LIN {X 0,Y 206.722,Z 761.527,A -85,B 0,C 180,E1 -21275.32,E2 -21275.32} C_VEL
LIN {X 0,Y 206.672,Z 761.479,A -85,B 0,C 180,E1 -21280.248,E2 -21280.248} C_VEL
LIN {X 0,Y 206.66,Z 761.554,A -85,B 0,C 180,E1 -21284.426,E2 -21284.426} C_VEL
LIN {X 0,Y 206.671,Z 761.526,A -85,B 0,C 180,E1 -21289.751,E2 -21289.751} C_VEL
LIN {X 0,Y 206.77,Z 761.618,A -85,B 0,C 180,E1 -21293.35,E2 -21293.35} C_VEL
LIN {X 0,Y 208.15,Z 768.058,A -85,B 0,C 180,E1 -21297.269,E2 -21297.269} C_VEL
LIN {X 0,Y 208.652,Z 770.291,A -85,B 0,C 180,E1 -21298.098,E2 -21298.098} C_VEL
LIN {X 0,Y 209.266,Z 773.35,A -85,B 0,C 180,E1 -21298.708,E2 -21298.708} C_VEL
LIN {X 0,Y 210.111,Z 778.796,A -85,B 0,C 180,E1 -21299.305,E2 -21299.305} C_VEL
LIN {X 0,Y 211.076,Z 793.394,A -85,B 0,C 180,E1 -21300.045,E2 -21300.045} C_VEL
LIN {X 0,Y 211.633,Z 797.547,A -85,B 0,C 180,E1 -21300.292,E2 -21300.292} C_VEL
LIN {X 0,Y 214.362,Z 818.731,A -85,B 0,C 180,E1 -21301.497,E2 -21301.497} C_VEL
LIN {X 0,Y 213.279,Z 848.564,A -85,B 0,C 180,E1 -21302.527,E2 -21302.527} C_VEL
LIN {X 0,Y 212.374,Z 858.849,A -85,B 0,C 180,E1 -21303.133,E2 -21303.133} C_VEL
LIN {X 0,Y 210.969,Z 869.629,A -85,B 0,C 180,E1 -21304.099,E2 -21304.099} C_VEL
LIN {X 0,Y 209.383,Z 879.305,A -85,B 0,C 180,E1 -21305.334,E2 -21305.334} C_VEL
LIN {X 0,Y 207.795,Z 887.072,A -85,B 0,C 180,E1 -21306.584,E2 -21306.584} C_VEL
LIN {X 0,Y 205.953,Z 895.137,A -85,B 0,C 180,E1 -21308.216,E2 -21308.216} C_VEL
LIN {X 0,Y 204.314,Z 901.802,A -85,B 0,C 180,E1 -21309.88,E2 -21309.88} C_VEL
LIN {X 0,Y 202.599,Z 908.13,A -85,B 0,C 180,E1 -21311.808,E2 -21311.808} C_VEL
LIN {X 0,Y 201.115,Z 913.389,A -85,B 0,C 180,E1 -21313.766,E2 -21313.766} C_VEL
LIN {X 0,Y 199.973,Z 917.78,A -85,B 0,C 180,E1 -21315.758,E2 -21315.758} C_VEL
LIN {X 0,Y 198.631,Z 922.961,A -85,B 0,C 180,E1 -21318.779,E2 -21318.779} C_VEL
LIN {X 0,Y 197.771,Z 926.768,A -85,B 0,C 180,E1 -21321.828,E2 -21321.828} C_VEL
LIN {X 0,Y 197.428,Z 928.517,A -85,B 0,C 180,E1 -21323.869,E2 -21323.869} C_VEL
LIN {X 0,Y 197.324,Z 929.773,A -85,B 0,C 180,E1 -21325.915,E2 -21325.915} C_VEL
LIN {X 0,Y 197.284,Z 930.553,A -85,B 0,C 180,E1 -21327.958,E2 -21327.958} C_VEL
LIN {X 0,Y 197.367,Z 930.849,A -85,B 0,C 180,E1 -21330,E2 -21330} C_VEL
LIN {X 0,Y 197.279,Z 930.544,A -85,B 0,C 180,E1 -21332.042,E2 -21332.042} C_VEL
LIN {X 0,Y 197.285,Z 929.748,A -85,B 0,C 180,E1 -21334.086,E2 -21334.086} C_VEL
LIN {X 0,Y 197.428,Z 928.477,A -85,B 0,C 180,E1 -21336.131,E2 -21336.131} C_VEL
LIN {X 0,Y 197.996,Z 925.55,A -85,B 0,C 180,E1 -21339.191,E2 -21339.191} C_VEL
LIN {X 0,Y 198.63,Z 922.885,A -85,B 0,C 180,E1 -21341.222,E2 -21341.222} C_VEL
LIN {X 0,Y 199.97,Z 917.682,A -85,B 0,C 180,E1 -21344.242,E2 -21344.242} C_VEL
LIN {X 0,Y 201.813,Z 910.825,A -85,B 0,C 180,E1 -21347.218,E2 -21347.218} C_VEL
LIN {X 0,Y 203.836,Z 903.341,A -85,B 0,C 180,E1 -21349.644,E2 -21349.644} C_VEL
LIN {X 0,Y 205.695,Z 895.961,A -85,B 0,C 180,E1 -21351.549,E2 -21351.549} C_VEL
LIN {X 0,Y 207.524,Z 888.058,A -85,B 0,C 180,E1 -21353.184,E2 -21353.184} C_VEL
LIN {X 0,Y 209.302,Z 879.229,A -85,B 0,C 180,E1 -21354.637,E2 -21354.637} C_VEL
LIN {X 0,Y 211.087,Z 868.011,A -85,B 0,C 180,E1 -21356.031,E2 -21356.031} C_VEL
LIN {X 0,Y 212.469,Z 857.353,A -85,B 0,C 180,E1 -21356.92,E2 -21356.92} C_VEL
LIN {X 0,Y 213.257,Z 847.507,A -85,B 0,C 180,E1 -21357.476,E2 -21357.476} C_VEL
LIN {X 0,Y 214.211,Z 817.801,A -85,B 0,C 180,E1 -21358.505,E2 -21358.505} C_VEL
LIN {X 0,Y 211.265,Z 795.967,A -85,B 0,C 180,E1 -21359.768,E2 -21359.768} C_VEL
LIN {X 0,Y 210.289,Z 791.346,A -85,B 0,C 180,E1 -21360.097,E2 -21360.097} C_VEL
LIN {X 0,Y 204.304,Z 777.141,A -85,B 0,C 180,E1 -21361.637,E2 -21361.637} C_VEL
LIN {X 0,Y 201.519,Z 770.64,A -85,B 0,C 180,E1 -21362.466,E2 -21362.466} C_VEL
LIN {X 0,Y 200.877,Z 767.771,A -85,B 0,C 180,E1 -21364.041,E2 -21364.041} C_VEL
LIN {X 0,Y 199.699,Z 762.434,A -85,B 0,C 180,E1 -21367.537,E2 -21367.537} C_VEL
LIN {X 0,Y 199.577,Z 762.407,A -85,B 0,C 180,E1 -21372.311,E2 -21372.311} C_VEL
LIN {X 0,Y 199.602,Z 762.436,A -85,B 0,C 180,E1 -21375.235,E2 -21375.235} C_VEL
LIN {X 0,Y 199.599,Z 762.38,A -85,B 0,C 180,E1 -21378.01,E2 -21378.01} C_VEL
LIN {X 0,Y 199.642,Z 762.35,A -85,B 0,C 180,E1 -21380.757,E2 -21380.757} C_VEL
LIN {X 0,Y 199.635,Z 762.425,A -85,B 0,C 180,E1 -21385.718,E2 -21385.718} C_VEL
LIN {X 0,Y 199.697,Z 762.416,A -85,B 0,C 180,E1 -21388.137,E2 -21388.137} C_VEL
LIN {X 0,Y 199.687,Z 762.415,A -85,B 0,C 180,E1 -21392.772,E2 -21392.772} C_VEL
LIN {X 0,Y 199.739,Z 762.391,A -85,B 0,C 180,E1 -21397.229,E2 -21397.229} C_VEL
LIN {X 0,Y 199.798,Z 762.404,A -85,B 0,C 180,E1 -21401.758,E2 -21401.758} C_VEL
LIN {X 0,Y 199.838,Z 762.381,A -85,B 0,C 180,E1 -21405.749,E2 -21405.749} C_VEL
LIN {X 0,Y 200.072,Z 762.355,A -85,B 0,C 180,E1 -21409.884,E2 -21409.884} C_VEL
LIN {X 0,Y 200.034,Z 762.375,A -85,B 0,C 180,E1 -21413.95,E2 -21413.95} C_VEL
LIN {X 0,Y 200.323,Z 762.303,A -85,B 0,C 180,E1 -21417.99,E2 -21417.99} C_VEL
LIN {X 0,Y 200.482,Z 762.304,A -85,B 0,C 180,E1 -21420,E2 -21420} C_VEL
LIN {X 0,Y 200.038,Z 762.373,A -85,B 0,C 180,E1 -21424.03,E2 -21424.03} C_VEL
LIN {X 0,Y 200.114,Z 762.33,A -85,B 0,C 180,E1 -21428.076,E2 -21428.076} C_VEL
LIN {X 0,Y 200.037,Z 762.367,A -85,B 0,C 180,E1 -21430.347,E2 -21430.347} C_VEL
LIN {X 0,Y 199.821,Z 762.398,A -85,B 0,C 180,E1 -21434.253,E2 -21434.253} C_VEL
LIN {X 0,Y 199.734,Z 762.388,A -85,B 0,C 180,E1 -21438.463,E2 -21438.463} C_VEL
LIN {X 0,Y 199.716,Z 762.405,A -85,B 0,C 180,E1 -21443.803,E2 -21443.803} C_VEL
LIN {X 0,Y 199.709,Z 762.413,A -85,B 0,C 180,E1 -21448.384,E2 -21448.384} C_VEL
LIN {X 0,Y 199.673,Z 762.406,A -85,B 0,C 180,E1 -21452.356,E2 -21452.356} C_VEL
LIN {X 0,Y 199.625,Z 762.432,A -85,B 0,C 180,E1 -21456.763,E2 -21456.763} C_VEL
LIN {X 0,Y 199.608,Z 762.402,A -85,B 0,C 180,E1 -21459.328,E2 -21459.328} C_VEL
LIN {X 0,Y 199.572,Z 762.367,A -85,B 0,C 180,E1 -21462.309,E2 -21462.309} C_VEL
LIN {X 0,Y 199.579,Z 762.394,A -85,B 0,C 180,E1 -21465.228,E2 -21465.228} C_VEL
LIN {X 0,Y 199.581,Z 762.438,A -85,B 0,C 180,E1 -21468.005,E2 -21468.005} C_VEL
LIN {X 0,Y 199.611,Z 762.396,A -85,B 0,C 180,E1 -21470.768,E2 -21470.768} C_VEL
LIN {X 0,Y 199.613,Z 762.433,A -85,B 0,C 180,E1 -21475.714,E2 -21475.714} C_VEL
LIN {X 0,Y 199.679,Z 762.569,A -85,B 0,C 180,E1 -21477.046,E2 -21477.046} C_VEL
LIN {X 0,Y 199.904,Z 763.577,A -85,B 0,C 180,E1 -21477.451,E2 -21477.451} C_VEL
LIN {X 0,Y 206.534,Z 775.877,A -85,B 0,C 180,E1 -21479.149,E2 -21479.149} C_VEL
LIN {X 0,Y 212.381,Z 789.676,A -85,B 0,C 180,E1 -21480.622,E2 -21480.622} C_VEL
LIN {X 0,Y 215.054,Z 797.212,A -85,B 0,C 180,E1 -21481.308,E2 -21481.308} C_VEL
LIN {X 0,Y 213.627,Z 837.05,A -85,B 0,C 180,E1 -21482.656,E2 -21482.656} C_VEL
LIN {X 0,Y 212.993,Z 846.207,A -85,B 0,C 180,E1 -21483.199,E2 -21483.199} C_VEL
LIN {X 0,Y 211.831,Z 856.411,A -85,B 0,C 180,E1 -21484.067,E2 -21484.067} C_VEL
LIN {X 0,Y 210.288,Z 866.725,A -85,B 0,C 180,E1 -21485.307,E2 -21485.307} C_VEL
LIN {X 0,Y 208.667,Z 875.367,A -85,B 0,C 180,E1 -21486.688,E2 -21486.688} C_VEL
LIN {X 0,Y 206.84,Z 883.481,A -85,B 0,C 180,E1 -21488.315,E2 -21488.315} C_VEL
LIN {X 0,Y 205.239,Z 890.171,A -85,B 0,C 180,E1 -21489.975,E2 -21489.975} C_VEL
LIN {X 0,Y 203.615,Z 896.506,A -85,B 0,C 180,E1 -21491.902,E2 -21491.902} C_VEL
LIN {X 0,Y 202.145,Z 901.771,A -85,B 0,C 180,E1 -21493.851,E2 -21493.851} C_VEL
LIN {X 0,Y 200.873,Z 906.166,A -85,B 0,C 180,E1 -21495.823,E2 -21495.823} C_VEL
LIN {X 0,Y 199.43,Z 911.33,A -85,B 0,C 180,E1 -21498.824,E2 -21498.824} C_VEL
LIN {X 0,Y 198.692,Z 913.977,A -85,B 0,C 180,E1 -21500.841,E2 -21500.841} C_VEL
LIN {X 0,Y 197.911,Z 916.875,A -85,B 0,C 180,E1 -21503.885,E2 -21503.885} C_VEL
LIN {X 0,Y 197.6,Z 918.137,A -85,B 0,C 180,E1 -21505.921,E2 -21505.921} C_VEL
LIN {X 0,Y 197.433,Z 918.931,A -85,B 0,C 180,E1 -21507.96,E2 -21507.96} C_VEL
LIN {X 0,Y 197.422,Z 919.232,A -85,B 0,C 180,E1 -21510,E2 -21510} C_VEL
LIN {X 0,Y 197.431,Z 918.953,A -85,B 0,C 180,E1 -21512.04,E2 -21512.04} C_VEL
LIN {X 0,Y 197.596,Z 918.204,A -85,B 0,C 180,E1 -21514.079,E2 -21514.079} C_VEL
LIN {X 0,Y 197.911,Z 916.987,A -85,B 0,C 180,E1 -21516.115,E2 -21516.115} C_VEL
LIN {X 0,Y 198.647,Z 914.137,A -85,B 0,C 180,E1 -21519.161,E2 -21519.161} C_VEL
LIN {X 0,Y 199.361,Z 911.54,A -85,B 0,C 180,E1 -21521.18,E2 -21521.18} C_VEL
LIN {X 0,Y 200.821,Z 906.431,A -85,B 0,C 180,E1 -21524.18,E2 -21524.18} C_VEL
LIN {X 0,Y 202.446,Z 900.93,A -85,B 0,C 180,E1 -21526.643,E2 -21526.643} C_VEL
LIN {X 0,Y 204.389,Z 894.011,A -85,B 0,C 180,E1 -21529.066,E2 -21529.066} C_VEL
LIN {X 0,Y 206.294,Z 886.068,A -85,B 0,C 180,E1 -21531.221,E2 -21531.221} C_VEL
LIN {X 0,Y 208.039,Z 878.489,A -85,B 0,C 180,E1 -21532.861,E2 -21532.861} C_VEL
LIN {X 0,Y 209.706,Z 870.538,A -85,B 0,C 180,E1 -21534.239,E2 -21534.239} C_VEL
LIN {X 0,Y 211.082,Z 862.32,A -85,B 0,C 180,E1 -21535.383,E2 -21535.383} C_VEL
LIN {X 0,Y 212.34,Z 853.505,A -85,B 0,C 180,E1 -21536.327,E2 -21536.327} C_VEL
LIN {X 0,Y 213.226,Z 844.156,A -85,B 0,C 180,E1 -21537.077,E2 -21537.077} C_VEL
LIN {X 0,Y 213.779,Z 835.371,A -85,B 0,C 180,E1 -21537.553,E2 -21537.553} C_VEL
LIN {X 0,Y 215.084,Z 797.029,A -85,B 0,C 180,E1 -21538.839,E2 -21538.839} C_VEL
LIN {X 0,Y 209.636,Z 782.862,A -85,B 0,C 180,E1 -21540.219,E2 -21540.219} C_VEL
LIN {X 0,Y 204.919,Z 772.617,A -85,B 0,C 180,E1 -21541.407,E2 -21541.407} C_VEL
LIN {X 0,Y 200.933,Z 765.668,A -85,B 0,C 180,E1 -21542.397,E2 -21542.397} C_VEL
LIN {X 0,Y 199.791,Z 763.102,A -85,B 0,C 180,E1 -21542.821,E2 -21542.821} C_VEL
LIN {X 0,Y 199.666,Z 762.492,A -85,B 0,C 180,E1 -21543.22,E2 -21543.22} C_VEL
LIN {X 0,Y 199.624,Z 762.403,A -85,B 0,C 180,E1 -21546.763,E2 -21546.763} C_VEL
LIN {X 0,Y 199.609,Z 762.395,A -85,B 0,C 180,E1 -21549.328,E2 -21549.328} C_VEL
LIN {X 0,Y 199.575,Z 762.439,A -85,B 0,C 180,E1 -21552.31,E2 -21552.31} C_VEL
LIN {X 0,Y 199.578,Z 762.388,A -85,B 0,C 180,E1 -21555.228,E2 -21555.228} C_VEL
LIN {X 0,Y 199.577,Z 762.368,A -85,B 0,C 180,E1 -21558.004,E2 -21558.004} C_VEL
LIN {X 0,Y 199.61,Z 762.4,A -85,B 0,C 180,E1 -21560.768,E2 -21560.768} C_VEL
LIN {X 0,Y 199.617,Z 762.431,A -85,B 0,C 180,E1 -21564.074,E2 -21564.074} C_VEL
LIN {X 0,Y 199.694,Z 762.407,A -85,B 0,C 180,E1 -21568.136,E2 -21568.136} C_VEL
LIN {X 0,Y 199.686,Z 762.402,A -85,B 0,C 180,E1 -21572.771,E2 -21572.771} C_VEL
LIN {X 0,Y 199.716,Z 762.415,A -85,B 0,C 180,E1 -21577.226,E2 -21577.226} C_VEL
LIN {X 0,Y 199.796,Z 762.38,A -85,B 0,C 180,E1 -21581.759,E2 -21581.759} C_VEL
LIN {X 0,Y 199.823,Z 762.396,A -85,B 0,C 180,E1 -21585.747,E2 -21585.747} C_VEL
LIN {X 0,Y 200.077,Z 762.359,A -85,B 0,C 180,E1 -21589.884,E2 -21589.884} C_VEL
LIN {X 0,Y 200.04,Z 762.347,A -85,B 0,C 180,E1 -21593.95,E2 -21593.95} C_VEL
LIN {X 0,Y 200.327,Z 762.341,A -85,B 0,C 180,E1 -21597.989,E2 -21597.989} C_VEL
LIN {X 0,Y 200.481,Z 762.305,A -85,B 0,C 180,E1 -21600,E2 -21600} C_VEL
LIN {X 0,Y 200.03,Z 762.35,A -85,B 0,C 180,E1 -21604.029,E2 -21604.029} C_VEL
LIN {X 0,Y 200.109,Z 762.369,A -85,B 0,C 180,E1 -21608.076,E2 -21608.076} C_VEL
LIN {X 0,Y 200.037,Z 762.356,A -85,B 0,C 180,E1 -21610.347,E2 -21610.347} C_VEL
LIN {X 0,Y 199.807,Z 762.409,A -85,B 0,C 180,E1 -21616.343,E2 -21616.343} C_VEL
LIN {X 0,Y 199.701,Z 762.391,A -85,B 0,C 180,E1 -21620.605,E2 -21620.605} C_VEL
LIN {X 0,Y 199.674,Z 762.424,A -85,B 0,C 180,E1 -21624.984,E2 -21624.984} C_VEL
LIN {X 0,Y 199.665,Z 762.4,A -85,B 0,C 180,E1 -21629.524,E2 -21629.524} C_VEL
LIN {X 0,Y 199.659,Z 762.425,A -85,B 0,C 180,E1 -21632.349,E2 -21632.349} C_VEL
LIN {X 0,Y 199.619,Z 762.377,A -85,B 0,C 180,E1 -21636.764,E2 -21636.764} C_VEL
LIN {X 0,Y 199.64,Z 762.35,A -85,B 0,C 180,E1 -21639.32,E2 -21639.32} C_VEL
LIN {X 0,Y 199.597,Z 762.39,A -85,B 0,C 180,E1 -21642.317,E2 -21642.317} C_VEL
LIN {X 0,Y 199.596,Z 762.435,A -85,B 0,C 180,E1 -21645.233,E2 -21645.233} C_VEL
LIN {X 0,Y 199.646,Z 762.413,A -85,B 0,C 180,E1 -21650.755,E2 -21650.755} C_VEL
LIN {X 0,Y 199.733,Z 762.619,A -85,B 0,C 180,E1 -21652.629,E2 -21652.629} C_VEL
LIN {X 0,Y 201.229,Z 769.521,A -85,B 0,C 180,E1 -21656.951,E2 -21656.951} C_VEL
LIN {X 0,Y 201.574,Z 770.95,A -85,B 0,C 180,E1 -21657.517,E2 -21657.517} C_VEL
LIN {X 0,Y 207.879,Z 785.226,A -85,B 0,C 180,E1 -21659.221,E2 -21659.221} C_VEL
LIN {X 0,Y 210.94,Z 793.406,A -85,B 0,C 180,E1 -21660.026,E2 -21660.026} C_VEL
LIN {X 0,Y 211.633,Z 797.547,A -85,B 0,C 180,E1 -21660.292,E2 -21660.292} C_VEL
LIN {X 0,Y 212.012,Z 803.342,A -85,B 0,C 180,E1 -21660.571,E2 -21660.571} C_VEL
LIN {X 0,Y 211.318,Z 809.241,A -85,B 0,C 180,E1 -21660.69,E2 -21660.69} C_VEL
LIN {X 0,Y 208.104,Z 825.054,A -85,B 0,C 180,E1 -21660.809,E2 -21660.809} C_VEL
LIN {X 0,Y 207.823,Z 829.057,A -85,B 0,C 180,E1 -21660.921,E2 -21660.921} C_VEL
LIN {X 0,Y 206.94,Z 849.591,A -85,B 0,C 180,E1 -21661.675,E2 -21661.675} C_VEL
LIN {X 0,Y 205.712,Z 861.756,A -85,B 0,C 180,E1 -21662.493,E2 -21662.493} C_VEL
LIN {X 0,Y 204.139,Z 872.294,A -85,B 0,C 180,E1 -21663.585,E2 -21663.585} C_VEL
LIN {X 0,Y 202.585,Z 880.857,A -85,B 0,C 180,E1 -21664.769,E2 -21664.769} C_VEL
LIN {X 0,Y 200.722,Z 889.329,A -85,B 0,C 180,E1 -21666.256,E2 -21666.256} C_VEL
LIN {X 0,Y 198.669,Z 898.002,A -85,B 0,C 180,E1 -21668.195,E2 -21668.195} C_VEL
LIN {X 0,Y 196.289,Z 906.5,A -85,B 0,C 180,E1 -21670.659,E2 -21670.659} C_VEL
LIN {X 0,Y 194.69,Z 912.006,A -85,B 0,C 180,E1 -21672.674,E2 -21672.674} C_VEL
LIN {X 0,Y 193.093,Z 917.572,A -85,B 0,C 180,E1 -21675.239,E2 -21675.239} C_VEL
LIN {X 0,Y 191.666,Z 922.753,A -85,B 0,C 180,E1 -21678.365,E2 -21678.365} C_VEL
LIN {X 0,Y 190.736,Z 926.559,A -85,B 0,C 180,E1 -21681.524,E2 -21681.524} C_VEL
LIN {X 0,Y 190.369,Z 928.309,A -85,B 0,C 180,E1 -21683.641,E2 -21683.641} C_VEL
LIN {X 0,Y 190.23,Z 929.651,A -85,B 0,C 180,E1 -21685.952,E2 -21685.952} C_VEL
LIN {X 0,Y 190.194,Z 930.344,A -85,B 0,C 180,E1 -21687.882,E2 -21687.882} C_VEL
LIN {X 0,Y 190.27,Z 930.641,A -85,B 0,C 180,E1 -21690,E2 -21690} C_VEL
LIN {X 0,Y 190.187,Z 930.336,A -85,B 0,C 180,E1 -21692.118,E2 -21692.118} C_VEL
LIN {X 0,Y 190.197,Z 929.538,A -85,B 0,C 180,E1 -21694.238,E2 -21694.238} C_VEL
LIN {X 0,Y 190.369,Z 928.267,A -85,B 0,C 180,E1 -21696.359,E2 -21696.359} C_VEL
LIN {X 0,Y 190.99,Z 925.34,A -85,B 0,C 180,E1 -21699.531,E2 -21699.531} C_VEL
LIN {X 0,Y 191.665,Z 922.675,A -85,B 0,C 180,E1 -21701.635,E2 -21701.635} C_VEL
LIN {X 0,Y 193.091,Z 917.471,A -85,B 0,C 180,E1 -21704.761,E2 -21704.761} C_VEL
LIN {X 0,Y 195.021,Z 910.613,A -85,B 0,C 180,E1 -21707.837,E2 -21707.837} C_VEL
LIN {X 0,Y 197.163,Z 903.13,A -85,B 0,C 180,E1 -21710.337,E2 -21710.337} C_VEL
LIN {X 0,Y 199.091,Z 895.749,A -85,B 0,C 180,E1 -21712.302,E2 -21712.302} C_VEL
LIN {X 0,Y 201.028,Z 887.846,A -85,B 0,C 180,E1 -21713.98,E2 -21713.98} C_VEL
LIN {X 0,Y 202.774,Z 879.515,A -85,B 0,C 180,E1 -21715.394,E2 -21715.394} C_VEL
LIN {X 0,Y 204.587,Z 868.8,A -85,B 0,C 180,E1 -21716.8,E2 -21716.8} C_VEL
LIN {X 0,Y 206.079,Z 857.957,A -85,B 0,C 180,E1 -21717.757,E2 -21717.757} C_VEL
LIN {X 0,Y 206.918,Z 848.581,A -85,B 0,C 180,E1 -21718.324,E2 -21718.324} C_VEL
LIN {X 0,Y 208.079,Z 820.343,A -85,B 0,C 180,E1 -21719.319,E2 -21719.319} C_VEL
LIN {X 0,Y 205.526,Z 799.524,A -85,B 0,C 180,E1 -21720.538,E2 -21720.538} C_VEL
LIN {X 0,Y 204.51,Z 794.28,A -85,B 0,C 180,E1 -21720.914,E2 -21720.914} C_VEL
LIN {X 0,Y 199.09,Z 781.161,A -85,B 0,C 180,E1 -21722.39,E2 -21722.39} C_VEL
LIN {X 0,Y 194.258,Z 770.481,A -85,B 0,C 180,E1 -21723.817,E2 -21723.817} C_VEL
LIN {X 0,Y 193.594,Z 767.517,A -85,B 0,C 180,E1 -21725.51,E2 -21725.51} C_VEL
LIN {X 0,Y 192.623,Z 763.317,A -85,B 0,C 180,E1 -21728.448,E2 -21728.448} C_VEL
LIN {X 0,Y 192.522,Z 763.306,A -85,B 0,C 180,E1 -21733.915,E2 -21733.915} C_VEL
LIN {X 0,Y 192.534,Z 763.244,A -85,B 0,C 180,E1 -21738.925,E2 -21738.925} C_VEL
LIN {X 0,Y 192.591,Z 763.255,A -85,B 0,C 180,E1 -21743.4,E2 -21743.4} C_VEL
LIN {X 0,Y 192.606,Z 763.307,A -85,B 0,C 180,E1 -21747.061,E2 -21747.061} C_VEL
LIN {X 0,Y 192.661,Z 763.277,A -85,B 0,C 180,E1 -21751.692,E2 -21751.692} C_VEL
LIN {X 0,Y 192.707,Z 763.278,A -85,B 0,C 180,E1 -21756.349,E2 -21756.349} C_VEL
LIN {X 0,Y 192.733,Z 763.282,A -85,B 0,C 180,E1 -21761.458,E2 -21761.458} C_VEL
LIN {X 0,Y 192.766,Z 763.268,A -85,B 0,C 180,E1 -21765.214,E2 -21765.214} C_VEL
LIN {X 0,Y 192.982,Z 763.232,A -85,B 0,C 180,E1 -21769.509,E2 -21769.509} C_VEL
LIN {X 0,Y 193.06,Z 763.246,A -85,B 0,C 180,E1 -21771.627,E2 -21771.627} C_VEL
LIN {X 0,Y 193.265,Z 763.181,A -85,B 0,C 180,E1 -21777.916,E2 -21777.916} C_VEL
LIN {X 0,Y 193.445,Z 763.179,A -85,B 0,C 180,E1 -21780,E2 -21780} C_VEL
LIN {X 0,Y 192.984,Z 763.25,A -85,B 0,C 180,E1 -21784.177,E2 -21784.177} C_VEL
LIN {X 0,Y 193.064,Z 763.209,A -85,B 0,C 180,E1 -21788.373,E2 -21788.373} C_VEL
LIN {X 0,Y 192.805,Z 763.282,A -85,B 0,C 180,E1 -21792.633,E2 -21792.633} C_VEL
LIN {X 0,Y 192.723,Z 763.255,A -85,B 0,C 180,E1 -21796.962,E2 -21796.962} C_VEL
LIN {X 0,Y 192.613,Z 763.305,A -85,B 0,C 180,E1 -21801.4,E2 -21801.4} C_VEL
LIN {X 0,Y 192.648,Z 763.279,A -85,B 0,C 180,E1 -21804.213,E2 -21804.213} C_VEL
LIN {X 0,Y 192.646,Z 763.297,A -85,B 0,C 180,E1 -21808.889,E2 -21808.889} C_VEL
LIN {X 0,Y 192.598,Z 763.283,A -85,B 0,C 180,E1 -21813.186,E2 -21813.186} C_VEL
LIN {X 0,Y 192.552,Z 763.3,A -85,B 0,C 180,E1 -21818.352,E2 -21818.352} C_VEL
LIN {X 0,Y 192.489,Z 763.25,A -85,B 0,C 180,E1 -21823.095,E2 -21823.095} C_VEL
LIN {X 0,Y 192.513,Z 763.312,A -85,B 0,C 180,E1 -21826.898,E2 -21826.898} C_VEL
LIN {X 0,Y 192.552,Z 763.271,A -85,B 0,C 180,E1 -21831.648,E2 -21831.648} C_VEL
LIN {X 0,Y 192.623,Z 763.519,A -85,B 0,C 180,E1 -21835.767,E2 -21835.767} C_VEL
LIN {X 0,Y 192.913,Z 764.719,A -85,B 0,C 180,E1 -21836.169,E2 -21836.169} C_VEL
LIN {X 0,Y 200.353,Z 777.936,A -85,B 0,C 180,E1 -21838.163,E2 -21838.163} C_VEL
LIN {X 0,Y 205.864,Z 790.701,A -85,B 0,C 180,E1 -21839.627,E2 -21839.627} C_VEL
LIN {X 0,Y 208.798,Z 798.726,A -85,B 0,C 180,E1 -21840.414,E2 -21840.414} C_VEL
LIN {X 0,Y 207.387,Z 836.648,A -85,B 0,C 180,E1 -21841.728,E2 -21841.728} C_VEL
LIN {X 0,Y 206.777,Z 845.79,A -85,B 0,C 180,E1 -21842.272,E2 -21842.272} C_VEL
LIN {X 0,Y 205.711,Z 855.078,A -85,B 0,C 180,E1 -21843.06,E2 -21843.06} C_VEL
LIN {X 0,Y 204.103,Z 865.258,A -85,B 0,C 180,E1 -21844.232,E2 -21844.232} C_VEL
LIN {X 0,Y 202.19,Z 875.579,A -85,B 0,C 180,E1 -21845.894,E2 -21845.894} C_VEL
LIN {X 0,Y 200.274,Z 883.693,A -85,B 0,C 180,E1 -21847.566,E2 -21847.566} C_VEL
LIN {X 0,Y 198.584,Z 890.383,A -85,B 0,C 180,E1 -21849.274,E2 -21849.274} C_VEL
LIN {X 0,Y 196.892,Z 896.717,A -85,B 0,C 180,E1 -21851.261,E2 -21851.261} C_VEL
LIN {X 0,Y 195.33,Z 901.982,A -85,B 0,C 180,E1 -21853.271,E2 -21853.271} C_VEL
LIN {X 0,Y 194.011,Z 906.376,A -85,B 0,C 180,E1 -21855.311,E2 -21855.311} C_VEL
LIN {X 0,Y 192.472,Z 911.54,A -85,B 0,C 180,E1 -21858.415,E2 -21858.415} C_VEL
LIN {X 0,Y 191.679,Z 914.187,A -85,B 0,C 180,E1 -21860.503,E2 -21860.503} C_VEL
LIN {X 0,Y 190.756,Z 917.447,A -85,B 0,C 180,E1 -21864.132,E2 -21864.132} C_VEL
LIN {X 0,Y 190.343,Z 919.14,A -85,B 0,C 180,E1 -21867.884,E2 -21867.884} C_VEL
LIN {X 0,Y 190.325,Z 919.441,A -85,B 0,C 180,E1 -21870,E2 -21870} C_VEL
LIN {X 0,Y 190.341,Z 919.162,A -85,B 0,C 180,E1 -21872.116,E2 -21872.116} C_VEL
LIN {X 0,Y 190.791,Z 917.479,A -85,B 0,C 180,E1 -21875.969,E2 -21875.969} C_VEL
LIN {X 0,Y 191.359,Z 915.488,A -85,B 0,C 180,E1 -21878.448,E2 -21878.448} C_VEL
LIN {X 0,Y 192.392,Z 911.748,A -85,B 0,C 180,E1 -21881.59,E2 -21881.59} C_VEL
LIN {X 0,Y 193.967,Z 906.638,A -85,B 0,C 180,E1 -21884.692,E2 -21884.692} C_VEL
LIN {X 0,Y 195.664,Z 901.136,A -85,B 0,C 180,E1 -21887.237,E2 -21887.237} C_VEL
LIN {X 0,Y 197.691,Z 894.217,A -85,B 0,C 180,E1 -21889.739,E2 -21889.739} C_VEL
LIN {X 0,Y 199.707,Z 886.273,A -85,B 0,C 180,E1 -21891.957,E2 -21891.957} C_VEL
LIN {X 0,Y 201.534,Z 878.694,A -85,B 0,C 180,E1 -21893.643,E2 -21893.643} C_VEL
LIN {X 0,Y 203.28,Z 870.741,A -85,B 0,C 180,E1 -21895.057,E2 -21895.057} C_VEL
LIN {X 0,Y 204.7,Z 862.522,A -85,B 0,C 180,E1 -21896.234,E2 -21896.234} C_VEL
LIN {X 0,Y 206.029,Z 853.549,A -85,B 0,C 180,E1 -21897.216,E2 -21897.216} C_VEL
LIN {X 0,Y 206.986,Z 843.711,A -85,B 0,C 180,E1 -21898.017,E2 -21898.017} C_VEL
LIN {X 0,Y 207.698,Z 832.427,A -85,B 0,C 180,E1 -21898.597,E2 -21898.597} C_VEL
LIN {X 0,Y 208.825,Z 798.59,A -85,B 0,C 180,E1 -21899.736,E2 -21899.736} C_VEL
LIN {X 0,Y 203.658,Z 785.218,A -85,B 0,C 180,E1 -21901.115,E2 -21901.115} C_VEL
LIN {X 0,Y 199.525,Z 776.327,A -85,B 0,C 180,E1 -21902.21,E2 -21902.21} C_VEL
LIN {X 0,Y 194.142,Z 766.942,A -85,B 0,C 180,E1 -21903.632,E2 -21903.632} C_VEL
LIN {X 0,Y 192.728,Z 764.096,A -85,B 0,C 180,E1 -21904.123,E2 -21904.123} C_VEL
LIN {X 0,Y 192.563,Z 763.365,A -85,B 0,C 180,E1 -21904.627,E2 -21904.627} C_VEL
LIN {X 0,Y 192.552,Z 763.271,A -85,B 0,C 180,E1 -21908.352,E2 -21908.352} C_VEL
LIN {X 0,Y 192.513,Z 763.315,A -85,B 0,C 180,E1 -21913.102,E2 -21913.102} C_VEL
LIN {X 0,Y 192.489,Z 763.251,A -85,B 0,C 180,E1 -21916.905,E2 -21916.905} C_VEL
LIN {X 0,Y 192.552,Z 763.298,A -85,B 0,C 180,E1 -21921.648,E2 -21921.648} C_VEL
LIN {X 0,Y 192.598,Z 763.283,A -85,B 0,C 180,E1 -21926.814,E2 -21926.814} C_VEL
LIN {X 0,Y 192.662,Z 763.29,A -85,B 0,C 180,E1 -21931.691,E2 -21931.691} C_VEL
LIN {X 0,Y 192.687,Z 763.281,A -85,B 0,C 180,E1 -21936.346,E2 -21936.346} C_VEL
LIN {X 0,Y 192.731,Z 763.262,A -85,B 0,C 180,E1 -21941.459,E2 -21941.459} C_VEL
LIN {X 0,Y 192.751,Z 763.272,A -85,B 0,C 180,E1 -21945.213,E2 -21945.213} C_VEL
LIN {X 0,Y 193.022,Z 763.242,A -85,B 0,C 180,E1 -21949.51,E2 -21949.51} C_VEL
LIN {X 0,Y 193.003,Z 763.22,A -85,B 0,C 180,E1 -21953.728,E2 -21953.728} C_VEL
LIN {X 0,Y 193.269,Z 763.221,A -85,B 0,C 180,E1 -21957.916,E2 -21957.916} C_VEL
LIN {X 0,Y 193.445,Z 763.18,A -85,B 0,C 180,E1 -21960,E2 -21960} C_VEL
LIN {X 0,Y 192.976,Z 763.229,A -85,B 0,C 180,E1 -21964.177,E2 -21964.177} C_VEL
LIN {X 0,Y 193.06,Z 763.246,A -85,B 0,C 180,E1 -21968.373,E2 -21968.373} C_VEL
LIN {X 0,Y 192.811,Z 763.242,A -85,B 0,C 180,E1 -21972.633,E2 -21972.633} C_VEL
LIN {X 0,Y 192.759,Z 763.286,A -85,B 0,C 180,E1 -21976.958,E2 -21976.958} C_VEL
LIN {X 0,Y 192.637,Z 763.268,A -85,B 0,C 180,E1 -21981.397,E2 -21981.397} C_VEL
LIN {X 0,Y 192.665,Z 763.291,A -85,B 0,C 180,E1 -21984.225,E2 -21984.225} C_VEL
LIN {X 0,Y 192.645,Z 763.275,A -85,B 0,C 180,E1 -21988.889,E2 -21988.889} C_VEL
LIN {X 0,Y 192.599,Z 763.307,A -85,B 0,C 180,E1 -21993.185,E2 -21993.185} C_VEL
LIN {X 0,Y 192.568,Z 763.233,A -85,B 0,C 180,E1 -21998.348,E2 -21998.348} C_VEL
LIN {X 0,Y 192.531,Z 763.287,A -85,B 0,C 180,E1 -22003.108,E2 -22003.108} C_VEL
LIN {X 0,Y 192.518,Z 763.292,A -85,B 0,C 180,E1 -22006.896,E2 -22006.896} C_VEL
LIN {X 0,Y 192.645,Z 763.434,A -85,B 0,C 180,E1 -22011.67,E2 -22011.67} C_VEL
LIN {X 0,Y 194.187,Z 770.212,A -85,B 0,C 180,E1 -22016.036,E2 -22016.036} C_VEL
LIN {X 0,Y 195.919,Z 774.183,A -85,B 0,C 180,E1 -22016.658,E2 -22016.658} C_VEL
LIN {X 0,Y 202.723,Z 789.62,A -85,B 0,C 180,E1 -22018.534,E2 -22018.534} C_VEL
LIN {X 0,Y 204.935,Z 795.371,A -85,B 0,C 180,E1 -22019.139,E2 -22019.139} C_VEL
LIN {X 0,Y 207.575,Z 814.318,A -85,B 0,C 180,E1 -22020.311,E2 -22020.311} C_VEL
LIN {X 0,Y 208.165,Z 820.897,A -85,B 0,C 180,E1 -22020.658,E2 -22020.658} C_VEL
LIN {X 0,Y 207.823,Z 829.057,A -85,B 0,C 180,E1 -22020.921,E2 -22020.921} C_VEL
LIN {X 0,Y 207.117,Z 834.914,A -85,B 0,C 180,E1 -22021.034,E2 -22021.034} C_VEL
LIN {X 0,Y 204.156,Z 844.404,A -85,B 0,C 180,E1 -22020.977,E2 -22020.977} C_VEL
LIN {X 0,Y 200.879,Z 853.784,A -85,B 0,C 180,E1 -22021.037,E2 -22021.037} C_VEL
LIN {X 0,Y 199.714,Z 859.464,A -85,B 0,C 180,E1 -22021.368,E2 -22021.368} C_VEL
LIN {X 0,Y 197.999,Z 870.919,A -85,B 0,C 180,E1 -22022.52,E2 -22022.52} C_VEL
LIN {X 0,Y 196.347,Z 879.974,A -85,B 0,C 180,E1 -22023.779,E2 -22023.779} C_VEL
LIN {X 0,Y 194.56,Z 887.894,A -85,B 0,C 180,E1 -22025.17,E2 -22025.17} C_VEL
LIN {X 0,Y 192.565,Z 895.748,A -85,B 0,C 180,E1 -22026.9,E2 -22026.9} C_VEL
LIN {X 0,Y 190.532,Z 903.097,A -85,B 0,C 180,E1 -22028.922,E2 -22028.922} C_VEL
LIN {X 0,Y 188.268,Z 910.553,A -85,B 0,C 180,E1 -22031.5,E2 -22031.5} C_VEL
LIN {X 0,Y 186.517,Z 916.403,A -85,B 0,C 180,E1 -22034.146,E2 -22034.146} C_VEL
LIN {X 0,Y 185.141,Z 921.018,A -85,B 0,C 180,E1 -22036.835,E2 -22036.835} C_VEL
LIN {X 0,Y 184.32,Z 924.02,A -85,B 0,C 180,E1 -22039.009,E2 -22039.009} C_VEL
LIN {X 0,Y 183.701,Z 926.351,A -85,B 0,C 180,E1 -22041.197,E2 -22041.197} C_VEL
LIN {X 0,Y 183.311,Z 928.101,A -85,B 0,C 180,E1 -22043.395,E2 -22043.395} C_VEL
LIN {X 0,Y 183.13,Z 929.621,A -85,B 0,C 180,E1 -22046.198,E2 -22046.198} C_VEL
LIN {X 0,Y 183.176,Z 930.432,A -85,B 0,C 180,E1 -22050,E2 -22050} C_VEL
LIN {X 0,Y 183.095,Z 929.669,A -85,B 0,C 180,E1 -22053.634,E2 -22053.634} C_VEL
LIN {X 0,Y 183.311,Z 928.057,A -85,B 0,C 180,E1 -22056.605,E2 -22056.605} C_VEL
LIN {X 0,Y 183.978,Z 925.13,A -85,B 0,C 180,E1 -22059.898,E2 -22059.898} C_VEL
LIN {X 0,Y 184.686,Z 922.464,A -85,B 0,C 180,E1 -22062.081,E2 -22062.081} C_VEL
LIN {X 0,Y 186.203,Z 917.26,A -85,B 0,C 180,E1 -22065.32,E2 -22065.32} C_VEL
LIN {X 0,Y 188.266,Z 910.402,A -85,B 0,C 180,E1 -22068.5,E2 -22068.5} C_VEL
LIN {X 0,Y 190.522,Z 902.918,A -85,B 0,C 180,E1 -22071.079,E2 -22071.079} C_VEL
LIN {X 0,Y 192.521,Z 895.536,A -85,B 0,C 180,E1 -22073.106,E2 -22073.106} C_VEL
LIN {X 0,Y 194.576,Z 887.634,A -85,B 0,C 180,E1 -22074.828,E2 -22074.828} C_VEL
LIN {X 0,Y 196.575,Z 878.447,A -85,B 0,C 180,E1 -22076.417,E2 -22076.417} C_VEL
LIN {X 0,Y 198.472,Z 867.452,A -85,B 0,C 180,E1 -22077.838,E2 -22077.838} C_VEL
LIN {X 0,Y 199.927,Z 856.907,A -85,B 0,C 180,E1 -22078.761,E2 -22078.761} C_VEL
LIN {X 0,Y 200.783,Z 847.059,A -85,B 0,C 180,E1 -22079.343,E2 -22079.343} C_VEL
LIN {X 0,Y 201.782,Z 819.471,A -85,B 0,C 180,E1 -22080.354,E2 -22080.354} C_VEL
LIN {X 0,Y 199.141,Z 799.112,A -85,B 0,C 180,E1 -22081.635,E2 -22081.635} C_VEL
LIN {X 0,Y 198.269,Z 795.792,A -85,B 0,C 180,E1 -22081.927,E2 -22081.927} C_VEL
LIN {X 0,Y 192.486,Z 781.943,A -85,B 0,C 180,E1 -22083.6,E2 -22083.6} C_VEL
LIN {X 0,Y 186.98,Z 770.228,A -85,B 0,C 180,E1 -22085.326,E2 -22085.326} C_VEL
LIN {X 0,Y 186.299,Z 767.258,A -85,B 0,C 180,E1 -22087.127,E2 -22087.127} C_VEL
LIN {X 0,Y 185.554,Z 764.221,A -85,B 0,C 180,E1 -22089.385,E2 -22089.385} C_VEL
LIN {X 0,Y 185.489,Z 764.181,A -85,B 0,C 180,E1 -22093.955,E2 -22093.955} C_VEL
LIN {X 0,Y 185.493,Z 764.116,A -85,B 0,C 180,E1 -22099.268,E2 -22099.268} C_VEL
LIN {X 0,Y 185.527,Z 764.121,A -85,B 0,C 180,E1 -22102.703,E2 -22102.703} C_VEL
LIN {X 0,Y 185.542,Z 764.18,A -85,B 0,C 180,E1 -22107.975,E2 -22107.975} C_VEL
LIN {X 0,Y 185.581,Z 764.153,A -85,B 0,C 180,E1 -22110.577,E2 -22110.577} C_VEL
LIN {X 0,Y 185.589,Z 764.175,A -85,B 0,C 180,E1 -22115.383,E2 -22115.383} C_VEL
LIN {X 0,Y 185.608,Z 764.151,A -85,B 0,C 180,E1 -22120.076,E2 -22120.076} C_VEL
LIN {X 0,Y 185.721,Z 764.154,A -85,B 0,C 180,E1 -22124.64,E2 -22124.64} C_VEL
LIN {X 0,Y 185.925,Z 764.108,A -85,B 0,C 180,E1 -22129.36,E2 -22129.36} C_VEL
LIN {X 0,Y 185.96,Z 764.132,A -85,B 0,C 180,E1 -22133.49,E2 -22133.49} C_VEL
LIN {X 0,Y 186.209,Z 764.06,A -85,B 0,C 180,E1 -22137.837,E2 -22137.837} C_VEL
LIN {X 0,Y 186.409,Z 764.054,A -85,B 0,C 180,E1 -22140,E2 -22140} C_VEL
LIN {X 0,Y 185.931,Z 764.126,A -85,B 0,C 180,E1 -22144.336,E2 -22144.336} C_VEL
LIN {X 0,Y 186.011,Z 764.089,A -85,B 0,C 180,E1 -22148.693,E2 -22148.693} C_VEL
LIN {X 0,Y 185.727,Z 764.161,A -85,B 0,C 180,E1 -22153.123,E2 -22153.123} C_VEL
LIN {X 0,Y 185.659,Z 764.135,A -85,B 0,C 180,E1 -22157.628,E2 -22157.628} C_VEL
LIN {X 0,Y 185.577,Z 764.181,A -85,B 0,C 180,E1 -22162.254,E2 -22162.254} C_VEL
LIN {X 0,Y 185.56,Z 764.157,A -85,B 0,C 180,E1 -22167.033,E2 -22167.033} C_VEL
LIN {X 0,Y 185.579,Z 764.182,A -85,B 0,C 180,E1 -22169.493,E2 -22169.493} C_VEL
LIN {X 0,Y 185.5,Z 764.172,A -85,B 0,C 180,E1 -22174.632,E2 -22174.632} C_VEL
LIN {X 0,Y 185.508,Z 764.189,A -85,B 0,C 180,E1 -22177.313,E2 -22177.313} C_VEL
LIN {X 0,Y 185.47,Z 764.133,A -85,B 0,C 180,E1 -22180.724,E2 -22180.724} C_VEL
LIN {X 0,Y 185.462,Z 764.166,A -85,B 0,C 180,E1 -22186.054,E2 -22186.054} C_VEL
LIN {X 0,Y 185.468,Z 764.163,A -85,B 0,C 180,E1 -22189.895,E2 -22189.895} C_VEL
LIN {X 0,Y 185.55,Z 764.381,A -85,B 0,C 180,E1 -22194.298,E2 -22194.298} C_VEL
LIN {X 0,Y 185.822,Z 765.574,A -85,B 0,C 180,E1 -22194.717,E2 -22194.717} C_VEL
LIN {X 0,Y 187.517,Z 768.345,A -85,B 0,C 180,E1 -22195.233,E2 -22195.233} C_VEL
LIN {X 0,Y 195.099,Z 781.817,A -85,B 0,C 180,E1 -22197.357,E2 -22197.357} C_VEL
LIN {X 0,Y 200.367,Z 794.202,A -85,B 0,C 180,E1 -22198.837,E2 -22198.837} C_VEL
LIN {X 0,Y 202.668,Z 800.6,A -85,B 0,C 180,E1 -22199.492,E2 -22199.492} C_VEL
LIN {X 0,Y 201.163,Z 837.041,A -85,B 0,C 180,E1 -22200.779,E2 -22200.779} C_VEL
LIN {X 0,Y 200.489,Z 846.158,A -85,B 0,C 180,E1 -22201.336,E2 -22201.336} C_VEL
LIN {X 0,Y 199.163,Z 857.114,A -85,B 0,C 180,E1 -22202.313,E2 -22202.313} C_VEL
LIN {X 0,Y 197.481,Z 867.152,A -85,B 0,C 180,E1 -22203.586,E2 -22203.586} C_VEL
LIN {X 0,Y 195.755,Z 875.791,A -85,B 0,C 180,E1 -22205.049,E2 -22205.049} C_VEL
LIN {X 0,Y 193.744,Z 883.905,A -85,B 0,C 180,E1 -22206.766,E2 -22206.766} C_VEL
LIN {X 0,Y 191.961,Z 890.595,A -85,B 0,C 180,E1 -22208.524,E2 -22208.524} C_VEL
LIN {X 0,Y 190.176,Z 896.928,A -85,B 0,C 180,E1 -22210.574,E2 -22210.574} C_VEL
LIN {X 0,Y 188.538,Z 902.193,A -85,B 0,C 180,E1 -22212.65,E2 -22212.65} C_VEL
LIN {X 0,Y 187.172,Z 906.586,A -85,B 0,C 180,E1 -22214.761,E2 -22214.761} C_VEL
LIN {X 0,Y 185.513,Z 911.751,A -85,B 0,C 180,E1 -22217.974,E2 -22217.974} C_VEL
LIN {X 0,Y 184.694,Z 914.397,A -85,B 0,C 180,E1 -22220.14,E2 -22220.14} C_VEL
LIN {X 0,Y 183.824,Z 917.294,A -85,B 0,C 180,E1 -22223.414,E2 -22223.414} C_VEL
LIN {X 0,Y 183.445,Z 918.556,A -85,B 0,C 180,E1 -22225.606,E2 -22225.606} C_VEL
LIN {X 0,Y 183.256,Z 919.349,A -85,B 0,C 180,E1 -22227.802,E2 -22227.802} C_VEL
LIN {X 0,Y 183.232,Z 919.65,A -85,B 0,C 180,E1 -22230,E2 -22230} C_VEL
LIN {X 0,Y 183.254,Z 919.371,A -85,B 0,C 180,E1 -22232.198,E2 -22232.198} C_VEL
LIN {X 0,Y 183.649,Z 918.005,A -85,B 0,C 180,E1 -22235.738,E2 -22235.738} C_VEL
LIN {X 0,Y 184.335,Z 915.696,A -85,B 0,C 180,E1 -22238.772,E2 -22238.772} C_VEL
LIN {X 0,Y 185.44,Z 911.955,A -85,B 0,C 180,E1 -22242.031,E2 -22242.031} C_VEL
LIN {X 0,Y 187.119,Z 906.845,A -85,B 0,C 180,E1 -22245.243,E2 -22245.243} C_VEL
LIN {X 0,Y 188.89,Z 901.344,A -85,B 0,C 180,E1 -22247.876,E2 -22247.876} C_VEL
LIN {X 0,Y 191.029,Z 894.423,A -85,B 0,C 180,E1 -22250.457,E2 -22250.457} C_VEL
LIN {X 0,Y 193.159,Z 886.478,A -85,B 0,C 180,E1 -22252.742,E2 -22252.742} C_VEL
LIN {X 0,Y 195.075,Z 878.898,A -85,B 0,C 180,E1 -22254.476,E2 -22254.476} C_VEL
LIN {X 0,Y 196.883,Z 870.945,A -85,B 0,C 180,E1 -22255.93,E2 -22255.93} C_VEL
LIN {X 0,Y 198.358,Z 862.725,A -85,B 0,C 180,E1 -22257.14,E2 -22257.14} C_VEL
LIN {X 0,Y 199.674,Z 854.394,A -85,B 0,C 180,E1 -22258.082,E2 -22258.082} C_VEL
LIN {X 0,Y 200.608,Z 845.575,A -85,B 0,C 180,E1 -22258.847,E2 -22258.847} C_VEL
LIN {X 0,Y 201.279,Z 836.35,A -85,B 0,C 180,E1 -22259.393,E2 -22259.393} C_VEL
LIN {X 0,Y 202.663,Z 800.28,A -85,B 0,C 180,E1 -22260.675,E2 -22260.675} C_VEL
LIN {X 0,Y 197.658,Z 787.418,A -85,B 0,C 180,E1 -22262.086,E2 -22262.086} C_VEL
LIN {X 0,Y 193.221,Z 778.153,A -85,B 0,C 180,E1 -22263.324,E2 -22263.324} C_VEL
LIN {X 0,Y 187.101,Z 767.858,A -85,B 0,C 180,E1 -22265.047,E2 -22265.047} C_VEL
LIN {X 0,Y 185.646,Z 764.909,A -85,B 0,C 180,E1 -22265.602,E2 -22265.602} C_VEL
LIN {X 0,Y 185.537,Z 764.239,A -85,B 0,C 180,E1 -22266.082,E2 -22266.082} C_VEL
LIN {X 0,Y 185.472,Z 764.169,A -85,B 0,C 180,E1 -22270.724,E2 -22270.724} C_VEL
LIN {X 0,Y 185.462,Z 764.17,A -85,B 0,C 180,E1 -22273.946,E2 -22273.946} C_VEL
LIN {X 0,Y 185.47,Z 764.132,A -85,B 0,C 180,E1 -22279.276,E2 -22279.276} C_VEL
LIN {X 0,Y 185.508,Z 764.188,A -85,B 0,C 180,E1 -22282.711,E2 -22282.711} C_VEL
LIN {X 0,Y 185.543,Z 764.167,A -85,B 0,C 180,E1 -22287.975,E2 -22287.975} C_VEL
LIN {X 0,Y 185.582,Z 764.182,A -85,B 0,C 180,E1 -22290.577,E2 -22290.577} C_VEL
LIN {X 0,Y 185.581,Z 764.154,A -85,B 0,C 180,E1 -22295.381,E2 -22295.381} C_VEL
LIN {X 0,Y 185.674,Z 764.143,A -85,B 0,C 180,E1 -22301.135,E2 -22301.135} C_VEL
LIN {X 0,Y 185.729,Z 764.161,A -85,B 0,C 180,E1 -22306.877,E2 -22306.877} C_VEL
LIN {X 0,Y 186.026,Z 764.088,A -85,B 0,C 180,E1 -22311.308,E2 -22311.308} C_VEL
LIN {X 0,Y 186.213,Z 764.1,A -85,B 0,C 180,E1 -22317.837,E2 -22317.837} C_VEL
LIN {X 0,Y 186.409,Z 764.055,A -85,B 0,C 180,E1 -22320,E2 -22320} C_VEL
LIN {X 0,Y 185.924,Z 764.109,A -85,B 0,C 180,E1 -22324.336,E2 -22324.336} C_VEL
LIN {X 0,Y 186.008,Z 764.123,A -85,B 0,C 180,E1 -22328.692,E2 -22328.692} C_VEL
LIN {X 0,Y 185.736,Z 764.125,A -85,B 0,C 180,E1 -22333.122,E2 -22333.122} C_VEL
LIN {X 0,Y 185.692,Z 764.165,A -85,B 0,C 180,E1 -22337.624,E2 -22337.624} C_VEL
LIN {X 0,Y 185.598,Z 764.148,A -85,B 0,C 180,E1 -22342.251,E2 -22342.251} C_VEL
LIN {X 0,Y 185.562,Z 764.174,A -85,B 0,C 180,E1 -22347.032,E2 -22347.032} C_VEL
LIN {X 0,Y 185.578,Z 764.153,A -85,B 0,C 180,E1 -22349.493,E2 -22349.493} C_VEL
LIN {X 0,Y 185.51,Z 764.177,A -85,B 0,C 180,E1 -22354.629,E2 -22354.629} C_VEL
LIN {X 0,Y 185.527,Z 764.12,A -85,B 0,C 180,E1 -22357.308,E2 -22357.308} C_VEL
LIN {X 0,Y 185.493,Z 764.117,A -85,B 0,C 180,E1 -22360.732,E2 -22360.732} C_VEL
LIN {X 0,Y 185.489,Z 764.179,A -85,B 0,C 180,E1 -22366.045,E2 -22366.045} C_VEL
LIN {X 0,Y 185.581,Z 764.324,A -85,B 0,C 180,E1 -22370.704,E2 -22370.704} C_VEL
LIN {X 0,Y 186.922,Z 770.018,A -85,B 0,C 180,E1 -22374.534,E2 -22374.534} C_VEL
LIN {X 0,Y 188.774,Z 774.052,A -85,B 0,C 180,E1 -22375.223,E2 -22375.223} C_VEL
LIN {X 0,Y 195.556,Z 788.899,A -85,B 0,C 180,E1 -22377.219,E2 -22377.219} C_VEL
LIN {X 0,Y 199.106,Z 798.325,A -85,B 0,C 180,E1 -22378.261,E2 -22378.261} C_VEL
LIN {X 0,Y 201.6,Z 817.2,A -85,B 0,C 180,E1 -22379.462,E2 -22379.462} C_VEL
LIN {X 0,Y 201.916,Z 822.532,A -85,B 0,C 180,E1 -22379.729,E2 -22379.729} C_VEL
LIN {X 0,Y 200.798,Z 848.178,A -85,B 0,C 180,E1 -22380.659,E2 -22380.659} C_VEL
LIN {X 0,Y 199.714,Z 859.464,A -85,B 0,C 180,E1 -22381.368,E2 -22381.368} C_VEL
LIN {X 0,Y 198.408,Z 865.05,A -85,B 0,C 180,E1 -22381.789,E2 -22381.789} C_VEL
LIN {X 0,Y 194.39,Z 873.879,A -85,B 0,C 180,E1 -22382.42,E2 -22382.42} C_VEL
LIN {X 0,Y 190.053,Z 882.305,A -85,B 0,C 180,E1 -22383.32,E2 -22383.32} C_VEL
LIN {X 0,Y 188.276,Z 887.179,A -85,B 0,C 180,E1 -22384.159,E2 -22384.159} C_VEL
LIN {X 0,Y 186.313,Z 894.519,A -85,B 0,C 180,E1 -22385.781,E2 -22385.781} C_VEL
LIN {X 0,Y 184.424,Z 901.182,A -85,B 0,C 180,E1 -22387.599,E2 -22387.599} C_VEL
LIN {X 0,Y 182.443,Z 907.509,A -85,B 0,C 180,E1 -22389.715,E2 -22389.715} C_VEL
LIN {X 0,Y 180.717,Z 912.767,A -85,B 0,C 180,E1 -22391.873,E2 -22391.873} C_VEL
LIN {X 0,Y 179.338,Z 917.156,A -85,B 0,C 180,E1 -22394.078,E2 -22394.078} C_VEL
LIN {X 0,Y 177.723,Z 922.336,A -85,B 0,C 180,E1 -22397.438,E2 -22397.438} C_VEL
LIN {X 0,Y 176.668,Z 926.142,A -85,B 0,C 180,E1 -22400.844,E2 -22400.844} C_VEL
LIN {X 0,Y 176.25,Z 927.892,A -85,B 0,C 180,E1 -22403.129,E2 -22403.129} C_VEL
LIN {X 0,Y 176.016,Z 929.633,A -85,B 0,C 180,E1 -22406.563,E2 -22406.563} C_VEL
LIN {X 0,Y 176.084,Z 930.223,A -85,B 0,C 180,E1 -22410,E2 -22410} C_VEL
LIN {X 0,Y 175.995,Z 929.656,A -85,B 0,C 180,E1 -22413.319,E2 -22413.319} C_VEL
LIN {X 0,Y 176.25,Z 927.848,A -85,B 0,C 180,E1 -22416.871,E2 -22416.871} C_VEL
LIN {X 0,Y 176.963,Z 924.92,A -85,B 0,C 180,E1 -22420.295,E2 -22420.295} C_VEL
LIN {X 0,Y 177.721,Z 922.253,A -85,B 0,C 180,E1 -22422.562,E2 -22422.562} C_VEL
LIN {X 0,Y 179.337,Z 917.049,A -85,B 0,C 180,E1 -22425.922,E2 -22425.922} C_VEL
LIN {X 0,Y 181.545,Z 910.191,A -85,B 0,C 180,E1 -22429.211,E2 -22429.211} C_VEL
LIN {X 0,Y 183.912,Z 902.707,A -85,B 0,C 180,E1 -22431.875,E2 -22431.875} C_VEL
LIN {X 0,Y 186.012,Z 895.324,A -85,B 0,C 180,E1 -22433.964,E2 -22433.964} C_VEL
LIN {X 0,Y 188.17,Z 887.422,A -85,B 0,C 180,E1 -22435.733,E2 -22435.733} C_VEL
LIN {X 0,Y 190.291,Z 878.005,A -85,B 0,C 180,E1 -22437.406,E2 -22437.406} C_VEL
LIN {X 0,Y 192.232,Z 867.236,A -85,B 0,C 180,E1 -22438.825,E2 -22438.825} C_VEL
LIN {X 0,Y 193.745,Z 856.688,A -85,B 0,C 180,E1 -22439.769,E2 -22439.769} C_VEL
LIN {X 0,Y 194.624,Z 846.834,A -85,B 0,C 180,E1 -22440.368,E2 -22440.368} C_VEL
LIN {X 0,Y 195.655,Z 820.257,A -85,B 0,C 180,E1 -22441.367,E2 -22441.367} C_VEL
LIN {X 0,Y 193.082,Z 800.006,A -85,B 0,C 180,E1 -22442.7,E2 -22442.7} C_VEL
LIN {X 0,Y 187.097,Z 785.39,A -85,B 0,C 180,E1 -22444.537,E2 -22444.537} C_VEL
LIN {X 0,Y 181.294,Z 773.436,A -85,B 0,C 180,E1 -22446.37,E2 -22446.37} C_VEL
LIN {X 0,Y 179.639,Z 769.762,A -85,B 0,C 180,E1 -22447.065,E2 -22447.065} C_VEL
LIN {X 0,Y 178.467,Z 765.181,A -85,B 0,C 180,E1 -22450.363,E2 -22450.363} C_VEL
LIN {X 0,Y 178.421,Z 765.074,A -85,B 0,C 180,E1 -22455.155,E2 -22455.155} C_VEL
LIN {X 0,Y 178.423,Z 765.005,A -85,B 0,C 180,E1 -22458.452,E2 -22458.452} C_VEL
LIN {X 0,Y 178.438,Z 765.022,A -85,B 0,C 180,E1 -22463.787,E2 -22463.787} C_VEL
LIN {X 0,Y 178.489,Z 765.065,A -85,B 0,C 180,E1 -22466.547,E2 -22466.547} C_VEL
LIN {X 0,Y 178.522,Z 765.033,A -85,B 0,C 180,E1 -22470.007,E2 -22470.007} C_VEL
LIN {X 0,Y 178.535,Z 765.058,A -85,B 0,C 180,E1 -22474.876,E2 -22474.876} C_VEL
LIN {X 0,Y 178.624,Z 765.028,A -85,B 0,C 180,E1 -22480.784,E2 -22480.784} C_VEL
LIN {X 0,Y 178.664,Z 765.038,A -85,B 0,C 180,E1 -22484.017,E2 -22484.017} C_VEL
LIN {X 0,Y 178.86,Z 764.985,A -85,B 0,C 180,E1 -22489.215,E2 -22489.215} C_VEL
LIN {X 0,Y 178.924,Z 765.009,A -85,B 0,C 180,E1 -22493.233,E2 -22493.233} C_VEL
LIN {X 0,Y 179.155,Z 764.938,A -85,B 0,C 180,E1 -22497.752,E2 -22497.752} C_VEL
LIN {X 0,Y 179.372,Z 764.93,A -85,B 0,C 180,E1 -22500,E2 -22500} C_VEL
LIN {X 0,Y 178.879,Z 765.003,A -85,B 0,C 180,E1 -22504.507,E2 -22504.507} C_VEL
LIN {X 0,Y 178.94,Z 764.972,A -85,B 0,C 180,E1 -22509.039,E2 -22509.039} C_VEL
LIN {X 0,Y 178.651,Z 765.041,A -85,B 0,C 180,E1 -22513.653,E2 -22513.653} C_VEL
LIN {X 0,Y 178.592,Z 765.027,A -85,B 0,C 180,E1 -22519.186,E2 -22519.186} C_VEL
LIN {X 0,Y 178.521,Z 765.03,A -85,B 0,C 180,E1 -22525.114,E2 -22525.114} C_VEL
LIN {X 0,Y 178.523,Z 765.06,A -85,B 0,C 180,E1 -22529.993,E2 -22529.993} C_VEL
LIN {X 0,Y 178.485,Z 765.042,A -85,B 0,C 180,E1 -22534.219,E2 -22534.219} C_VEL
LIN {X 0,Y 178.395,Z 765.043,A -85,B 0,C 180,E1 -22539.075,E2 -22539.075} C_VEL
LIN {X 0,Y 178.398,Z 765.003,A -85,B 0,C 180,E1 -22542.046,E2 -22542.046} C_VEL
LIN {X 0,Y 178.395,Z 765.025,A -85,B 0,C 180,E1 -22545.164,E2 -22545.164} C_VEL
LIN {X 0,Y 178.408,Z 765.065,A -85,B 0,C 180,E1 -22548.458,E2 -22548.458} C_VEL
LIN {X 0,Y 178.512,Z 765.256,A -85,B 0,C 180,E1 -22552.686,E2 -22552.686} C_VEL
LIN {X 0,Y 178.715,Z 766.212,A -85,B 0,C 180,E1 -22553.09,E2 -22553.09} C_VEL
LIN {X 0,Y 180.256,Z 768.96,A -85,B 0,C 180,E1 -22553.63,E2 -22553.63} C_VEL
LIN {X 0,Y 186.93,Z 780.17,A -85,B 0,C 180,E1 -22555.649,E2 -22555.649} C_VEL
LIN {X 0,Y 191.188,Z 788.526,A -85,B 0,C 180,E1 -22556.893,E2 -22556.893} C_VEL
LIN {X 0,Y 196.232,Z 801.398,A -85,B 0,C 180,E1 -22558.401,E2 -22558.401} C_VEL
LIN {X 0,Y 196.497,Z 803.436,A -85,B 0,C 180,E1 -22558.535,E2 -22558.535} C_VEL
LIN {X 0,Y 194.999,Z 837.371,A -85,B 0,C 180,E1 -22559.767,E2 -22559.767} C_VEL
LIN {X 0,Y 194.28,Z 846.527,A -85,B 0,C 180,E1 -22560.344,E2 -22560.344} C_VEL
LIN {X 0,Y 193.086,Z 856.135,A -85,B 0,C 180,E1 -22561.216,E2 -22561.216} C_VEL
LIN {X 0,Y 191.156,Z 867.366,A -85,B 0,C 180,E1 -22562.64,E2 -22562.64} C_VEL
LIN {X 0,Y 189.367,Z 876.003,A -85,B 0,C 180,E1 -22564.146,E2 -22564.146} C_VEL
LIN {X 0,Y 187.258,Z 884.116,A -85,B 0,C 180,E1 -22565.911,E2 -22565.911} C_VEL
LIN {X 0,Y 185.381,Z 890.806,A -85,B 0,C 180,E1 -22567.721,E2 -22567.721} C_VEL
LIN {X 0,Y 183.493,Z 897.14,A -85,B 0,C 180,E1 -22569.836,E2 -22569.836} C_VEL
LIN {X 0,Y 181.778,Z 902.404,A -85,B 0,C 180,E1 -22571.983,E2 -22571.983} C_VEL
LIN {X 0,Y 180.349,Z 906.795,A -85,B 0,C 180,E1 -22574.17,E2 -22574.17} C_VEL
LIN {X 0,Y 178.573,Z 911.961,A -85,B 0,C 180,E1 -22577.499,E2 -22577.499} C_VEL
LIN {X 0,Y 177.696,Z 914.607,A -85,B 0,C 180,E1 -22579.748,E2 -22579.748} C_VEL
LIN {X 0,Y 176.773,Z 917.503,A -85,B 0,C 180,E1 -22583.15,E2 -22583.15} C_VEL
LIN {X 0,Y 176.39,Z 918.764,A -85,B 0,C 180,E1 -22585.429,E2 -22585.429} C_VEL
LIN {X 0,Y 176.172,Z 919.558,A -85,B 0,C 180,E1 -22587.714,E2 -22587.714} C_VEL
LIN {X 0,Y 176.14,Z 919.859,A -85,B 0,C 180,E1 -22590,E2 -22590} C_VEL
LIN {X 0,Y 176.17,Z 919.579,A -85,B 0,C 180,E1 -22592.286,E2 -22592.286} C_VEL
LIN {X 0,Y 176.5,Z 918.46,A -85,B 0,C 180,E1 -22595.454,E2 -22595.454} C_VEL
LIN {X 0,Y 177.319,Z 915.904,A -85,B 0,C 180,E1 -22599.122,E2 -22599.122} C_VEL
LIN {X 0,Y 178.513,Z 912.163,A -85,B 0,C 180,E1 -22602.506,E2 -22602.506} C_VEL
LIN {X 0,Y 180.279,Z 907.052,A -85,B 0,C 180,E1 -22605.836,E2 -22605.836} C_VEL
LIN {X 0,Y 182.146,Z 901.55,A -85,B 0,C 180,E1 -22608.561,E2 -22608.561} C_VEL
LIN {X 0,Y 184.403,Z 894.629,A -85,B 0,C 180,E1 -22611.227,E2 -22611.227} C_VEL
LIN {X 0,Y 186.653,Z 886.683,A -85,B 0,C 180,E1 -22613.582,E2 -22613.582} C_VEL
LIN {X 0,Y 188.661,Z 879.102,A -85,B 0,C 180,E1 -22615.366,E2 -22615.366} C_VEL
LIN {X 0,Y 190.54,Z 871.148,A -85,B 0,C 180,E1 -22616.862,E2 -22616.862} C_VEL
LIN {X 0,Y 192.081,Z 862.927,A -85,B 0,C 180,E1 -22618.104,E2 -22618.104} C_VEL
LIN {X 0,Y 193.363,Z 855.236,A -85,B 0,C 180,E1 -22619.005,E2 -22619.005} C_VEL
LIN {X 0,Y 194.477,Z 845.349,A -85,B 0,C 180,E1 -22619.885,E2 -22619.885} C_VEL
LIN {X 0,Y 195.149,Z 836.466,A -85,B 0,C 180,E1 -22620.416,E2 -22620.416} C_VEL
LIN {X 0,Y 196.531,Z 801.981,A -85,B 0,C 180,E1 -22621.678,E2 -22621.678} C_VEL
LIN {X 0,Y 191.562,Z 789.337,A -85,B 0,C 180,E1 -22623.16,E2 -22623.16} C_VEL
LIN {X 0,Y 188.011,Z 782.098,A -85,B 0,C 180,E1 -22624.203,E2 -22624.203} C_VEL
LIN {X 0,Y 182.246,Z 772.277,A -85,B 0,C 180,E1 -22625.92,E2 -22625.92} C_VEL
LIN {X 0,Y 180.147,Z 768.825,A -85,B 0,C 180,E1 -22626.577,E2 -22626.577} C_VEL
LIN {X 0,Y 178.662,Z 765.973,A -85,B 0,C 180,E1 -22627.141,E2 -22627.141} C_VEL
LIN {X 0,Y 178.451,Z 765.155,A -85,B 0,C 180,E1 -22627.657,E2 -22627.657} C_VEL
LIN {X 0,Y 178.408,Z 765.072,A -85,B 0,C 180,E1 -22632.042,E2 -22632.042} C_VEL
LIN {X 0,Y 178.394,Z 765.023,A -85,B 0,C 180,E1 -22635.164,E2 -22635.164} C_VEL
LIN {X 0,Y 178.403,Z 765.004,A -85,B 0,C 180,E1 -22638.46,E2 -22638.46} C_VEL
LIN {X 0,Y 178.424,Z 765.073,A -85,B 0,C 180,E1 -22643.783,E2 -22643.783} C_VEL
LIN {X 0,Y 178.487,Z 765.04,A -85,B 0,C 180,E1 -22646.546,E2 -22646.546} C_VEL
LIN {X 0,Y 178.523,Z 765.06,A -85,B 0,C 180,E1 -22650.007,E2 -22650.007} C_VEL
LIN {X 0,Y 178.521,Z 765.03,A -85,B 0,C 180,E1 -22654.886,E2 -22654.886} C_VEL
LIN {X 0,Y 178.622,Z 765.025,A -85,B 0,C 180,E1 -22660.786,E2 -22660.786} C_VEL
LIN {X 0,Y 178.655,Z 765.039,A -85,B 0,C 180,E1 -22666.347,E2 -22666.347} C_VEL
LIN {X 0,Y 178.975,Z 764.968,A -85,B 0,C 180,E1 -22670.963,E2 -22670.963} C_VEL
LIN {X 0,Y 179.158,Z 764.979,A -85,B 0,C 180,E1 -22677.752,E2 -22677.752} C_VEL
LIN {X 0,Y 179.372,Z 764.93,A -85,B 0,C 180,E1 -22680,E2 -22680} C_VEL
LIN {X 0,Y 178.872,Z 764.989,A -85,B 0,C 180,E1 -22684.507,E2 -22684.507} C_VEL
LIN {X 0,Y 178.959,Z 764.996,A -85,B 0,C 180,E1 -22689.038,E2 -22689.038} C_VEL
LIN {X 0,Y 178.668,Z 765.009,A -85,B 0,C 180,E1 -22693.651,E2 -22693.651} C_VEL
LIN {X 0,Y 178.651,Z 765.037,A -85,B 0,C 180,E1 -22698.343,E2 -22698.343} C_VEL
LIN {X 0,Y 178.512,Z 765.038,A -85,B 0,C 180,E1 -22703.185,E2 -22703.185} C_VEL
LIN {X 0,Y 178.486,Z 765.041,A -85,B 0,C 180,E1 -22708.197,E2 -22708.197} C_VEL
LIN {X 0,Y 178.477,Z 765.044,A -85,B 0,C 180,E1 -22710.791,E2 -22710.791} C_VEL
LIN {X 0,Y 178.491,Z 765.058,A -85,B 0,C 180,E1 -22714.222,E2 -22714.222} C_VEL
LIN {X 0,Y 178.416,Z 764.99,A -85,B 0,C 180,E1 -22719.069,E2 -22719.069} C_VEL
LIN {X 0,Y 178.421,Z 765.015,A -85,B 0,C 180,E1 -22722.038,E2 -22722.038} C_VEL
LIN {X 0,Y 178.419,Z 765.073,A -85,B 0,C 180,E1 -22725.155,E2 -22725.155} C_VEL
LIN {X 0,Y 178.492,Z 765.246,A -85,B 0,C 180,E1 -22729.645,E2 -22729.645} C_VEL
LIN {X 0,Y 179.647,Z 769.81,A -85,B 0,C 180,E1 -22732.873,E2 -22732.873} C_VEL
LIN {X 0,Y 181.545,Z 773.804,A -85,B 0,C 180,E1 -22733.622,E2 -22733.622} C_VEL
LIN {X 0,Y 187.878,Z 787.096,A -85,B 0,C 180,E1 -22735.627,E2 -22735.627} C_VEL
LIN {X 0,Y 193.136,Z 800.152,A -85,B 0,C 180,E1 -22737.246,E2 -22737.246} C_VEL
LIN {X 0,Y 195.211,Z 815.247,A -85,B 0,C 180,E1 -22738.275,E2 -22738.275} C_VEL
LIN {X 0,Y 195.808,Z 822.345,A -85,B 0,C 180,E1 -22738.68,E2 -22738.68} C_VEL
LIN {X 0,Y 194.644,Z 847.985,A -85,B 0,C 180,E1 -22739.636,E2 -22739.636} C_VEL
LIN {X 0,Y 193.545,Z 859.077,A -85,B 0,C 180,E1 -22740.347,E2 -22740.347} C_VEL
LIN {X 0,Y 191.723,Z 870.716,A -85,B 0,C 180,E1 -22741.54,E2 -22741.54} C_VEL
LIN {X 0,Y 190.145,Z 879.153,A -85,B 0,C 180,E1 -22742.733,E2 -22742.733} C_VEL
LIN {X 0,Y 188.276,Z 887.179,A -85,B 0,C 180,E1 -22744.159,E2 -22744.159} C_VEL
LIN {X 0,Y 186.475,Z 892.023,A -85,B 0,C 180,E1 -22745.09,E2 -22745.09} C_VEL
LIN {X 0,Y 181.737,Z 899.335,A -85,B 0,C 180,E1 -22746.635,E2 -22746.635} C_VEL
LIN {X 0,Y 176.964,Z 905.883,A -85,B 0,C 180,E1 -22748.433,E2 -22748.433} C_VEL
LIN {X 0,Y 175.072,Z 909.501,A -85,B 0,C 180,E1 -22749.773,E2 -22749.773} C_VEL
LIN {X 0,Y 172.838,Z 915.986,A -85,B 0,C 180,E1 -22752.854,E2 -22752.854} C_VEL
LIN {X 0,Y 171.288,Z 920.601,A -85,B 0,C 180,E1 -22755.748,E2 -22755.748} C_VEL
LIN {X 0,Y 170.357,Z 923.603,A -85,B 0,C 180,E1 -22758.096,E2 -22758.096} C_VEL
LIN {X 0,Y 169.656,Z 925.934,A -85,B 0,C 180,E1 -22760.462,E2 -22760.462} C_VEL
LIN {X 0,Y 169.184,Z 927.683,A -85,B 0,C 180,E1 -22762.841,E2 -22762.841} C_VEL
LIN {X 0,Y 168.929,Z 929.576,A -85,B 0,C 180,E1 -22766.837,E2 -22766.837} C_VEL
LIN {X 0,Y 168.994,Z 930.014,A -85,B 0,C 180,E1 -22770,E2 -22770} C_VEL
LIN {X 0,Y 168.909,Z 929.591,A -85,B 0,C 180,E1 -22773.043,E2 -22773.043} C_VEL
LIN {X 0,Y 169.184,Z 927.638,A -85,B 0,C 180,E1 -22777.159,E2 -22777.159} C_VEL
LIN {X 0,Y 169.968,Z 924.709,A -85,B 0,C 180,E1 -22780.724,E2 -22780.724} C_VEL
LIN {X 0,Y 170.774,Z 922.042,A -85,B 0,C 180,E1 -22783.082,E2 -22783.082} C_VEL
LIN {X 0,Y 172.494,Z 916.838,A -85,B 0,C 180,E1 -22786.571,E2 -22786.571} C_VEL
LIN {X 0,Y 174.857,Z 909.98,A -85,B 0,C 180,E1 -22789.977,E2 -22789.977} C_VEL
LIN {X 0,Y 177.339,Z 902.495,A -85,B 0,C 180,E1 -22792.73,E2 -22792.73} C_VEL
LIN {X 0,Y 179.554,Z 895.112,A -85,B 0,C 180,E1 -22794.883,E2 -22794.883} C_VEL
LIN {X 0,Y 181.803,Z 887.209,A -85,B 0,C 180,E1 -22796.705,E2 -22796.705} C_VEL
LIN {X 0,Y 184.023,Z 877.792,A -85,B 0,C 180,E1 -22798.423,E2 -22798.423} C_VEL
LIN {X 0,Y 186.046,Z 867.02,A -85,B 0,C 180,E1 -22799.879,E2 -22799.879} C_VEL
LIN {X 0,Y 187.616,Z 856.469,A -85,B 0,C 180,E1 -22800.846,E2 -22800.846} C_VEL
LIN {X 0,Y 188.548,Z 846.61,A -85,B 0,C 180,E1 -22801.456,E2 -22801.456} C_VEL
LIN {X 0,Y 189.593,Z 821.055,A -85,B 0,C 180,E1 -22802.446,E2 -22802.446} C_VEL
LIN {X 0,Y 187.307,Z 802.546,A -85,B 0,C 180,E1 -22803.717,E2 -22803.717} C_VEL
LIN {X 0,Y 181.803,Z 788.952,A -85,B 0,C 180,E1 -22805.514,E2 -22805.514} C_VEL
LIN {X 0,Y 176.492,Z 777.752,A -85,B 0,C 180,E1 -22807.301,E2 -22807.301} C_VEL
LIN {X 0,Y 172.376,Z 769.732,A -85,B 0,C 180,E1 -22808.845,E2 -22808.845} C_VEL
LIN {X 0,Y 171.56,Z 766.716,A -85,B 0,C 180,E1 -22810.953,E2 -22810.953} C_VEL
LIN {X 0,Y 171.386,Z 766.024,A -85,B 0,C 180,E1 -22811.61,E2 -22811.61} C_VEL
LIN {X 0,Y 171.356,Z 765.898,A -85,B 0,C 180,E1 -22817.583,E2 -22817.583} C_VEL
LIN {X 0,Y 171.404,Z 765.869,A -85,B 0,C 180,E1 -22822.046,E2 -22822.046} C_VEL
LIN {X 0,Y 171.403,Z 765.928,A -85,B 0,C 180,E1 -22825.09,E2 -22825.09} C_VEL
LIN {X 0,Y 171.448,Z 765.913,A -85,B 0,C 180,E1 -22830.534,E2 -22830.534} C_VEL
LIN {X 0,Y 171.458,Z 765.93,A -85,B 0,C 180,E1 -22835.802,E2 -22835.802} C_VEL
LIN {X 0,Y 171.58,Z 765.906,A -85,B 0,C 180,E1 -22840.872,E2 -22840.872} C_VEL
LIN {X 0,Y 171.595,Z 765.895,A -85,B 0,C 180,E1 -22845.775,E2 -22845.775} C_VEL
LIN {X 0,Y 171.888,Z 765.872,A -85,B 0,C 180,E1 -22850.587,E2 -22850.587} C_VEL
LIN {X 0,Y 171.821,Z 765.868,A -85,B 0,C 180,E1 -22855.308,E2 -22855.308} C_VEL
LIN {X 0,Y 172.335,Z 765.805,A -85,B 0,C 180,E1 -22860,E2 -22860} C_VEL
LIN {X 0,Y 171.828,Z 765.877,A -85,B 0,C 180,E1 -22864.692,E2 -22864.692} C_VEL
LIN {X 0,Y 171.874,Z 765.855,A -85,B 0,C 180,E1 -22869.414,E2 -22869.414} C_VEL
LIN {X 0,Y 171.565,Z 765.915,A -85,B 0,C 180,E1 -22874.228,E2 -22874.228} C_VEL
LIN {X 0,Y 171.517,Z 765.912,A -85,B 0,C 180,E1 -22879.535,E2 -22879.535} C_VEL
LIN {X 0,Y 171.459,Z 765.907,A -85,B 0,C 180,E1 -22885.609,E2 -22885.609} C_VEL
LIN {X 0,Y 171.441,Z 765.939,A -85,B 0,C 180,E1 -22890.586,E2 -22890.586} C_VEL
LIN {X 0,Y 171.394,Z 765.931,A -85,B 0,C 180,E1 -22895.035,E2 -22895.035} C_VEL
LIN {X 0,Y 171.358,Z 765.923,A -85,B 0,C 180,E1 -22898.807,E2 -22898.807} C_VEL
LIN {X 0,Y 171.321,Z 765.891,A -85,B 0,C 180,E1 -22904.218,E2 -22904.218} C_VEL
LIN {X 0,Y 171.339,Z 765.934,A -85,B 0,C 180,E1 -22908.983,E2 -22908.983} C_VEL
LIN {X 0,Y 171.414,Z 766.232,A -85,B 0,C 180,E1 -22910.957,E2 -22910.957} C_VEL
LIN {X 0,Y 171.715,Z 767.351,A -85,B 0,C 180,E1 -22911.377,E2 -22911.377} C_VEL
LIN {X 0,Y 173.25,Z 769.87,A -85,B 0,C 180,E1 -22911.936,E2 -22911.936} C_VEL
LIN {X 0,Y 174.57,Z 772.021,A -85,B 0,C 180,E1 -22912.388,E2 -22912.388} C_VEL
LIN {X 0,Y 180.338,Z 781.499,A -85,B 0,C 180,E1 -22914.256,E2 -22914.256} C_VEL
LIN {X 0,Y 185.646,Z 791.555,A -85,B 0,C 180,E1 -22915.899,E2 -22915.899} C_VEL
LIN {X 0,Y 190.426,Z 803.894,A -85,B 0,C 180,E1 -22917.42,E2 -22917.42} C_VEL
LIN {X 0,Y 188.914,Z 837.159,A -85,B 0,C 180,E1 -22918.659,E2 -22918.659} C_VEL
LIN {X 0,Y 188.25,Z 846.093,A -85,B 0,C 180,E1 -22919.232,E2 -22919.232} C_VEL
LIN {X 0,Y 187.027,Z 855.641,A -85,B 0,C 180,E1 -22920.1,E2 -22920.1} C_VEL
LIN {X 0,Y 185.195,Z 865.901,A -85,B 0,C 180,E1 -22921.373,E2 -22921.373} C_VEL
LIN {X 0,Y 183.028,Z 876.215,A -85,B 0,C 180,E1 -22923.18,E2 -22923.18} C_VEL
LIN {X 0,Y 180.822,Z 884.328,A -85,B 0,C 180,E1 -22924.996,E2 -22924.996} C_VEL
LIN {X 0,Y 178.846,Z 891.017,A -85,B 0,C 180,E1 -22926.861,E2 -22926.861} C_VEL
LIN {X 0,Y 176.845,Z 897.351,A -85,B 0,C 180,E1 -22929.043,E2 -22929.043} C_VEL
LIN {X 0,Y 175.051,Z 902.614,A -85,B 0,C 180,E1 -22931.265,E2 -22931.265} C_VEL
LIN {X 0,Y 173.525,Z 907.006,A -85,B 0,C 180,E1 -22933.53,E2 -22933.53} C_VEL
LIN {X 0,Y 171.659,Z 912.171,A -85,B 0,C 180,E1 -22936.987,E2 -22936.987} C_VEL
LIN {X 0,Y 170.72,Z 914.817,A -85,B 0,C 180,E1 -22939.324,E2 -22939.324} C_VEL
LIN {X 0,Y 169.738,Z 917.712,A -85,B 0,C 180,E1 -22942.865,E2 -22942.865} C_VEL
LIN {X 0,Y 169.326,Z 918.973,A -85,B 0,C 180,E1 -22945.238,E2 -22945.238} C_VEL
LIN {X 0,Y 169.09,Z 919.766,A -85,B 0,C 180,E1 -22947.618,E2 -22947.618} C_VEL
LIN {X 0,Y 169.051,Z 920.067,A -85,B 0,C 180,E1 -22950,E2 -22950} C_VEL
LIN {X 0,Y 169.088,Z 919.787,A -85,B 0,C 180,E1 -22952.382,E2 -22952.382} C_VEL
LIN {X 0,Y 169.396,Z 918.822,A -85,B 0,C 180,E1 -22955.296,E2 -22955.296} C_VEL
LIN {X 0,Y 170.304,Z 916.112,A -85,B 0,C 180,E1 -22959.501,E2 -22959.501} C_VEL
LIN {X 0,Y 171.605,Z 912.37,A -85,B 0,C 180,E1 -22963.018,E2 -22963.018} C_VEL
LIN {X 0,Y 173.447,Z 907.26,A -85,B 0,C 180,E1 -22966.477,E2 -22966.477} C_VEL
LIN {X 0,Y 175.438,Z 901.757,A -85,B 0,C 180,E1 -22969.299,E2 -22969.299} C_VEL
LIN {X 0,Y 177.818,Z 894.835,A -85,B 0,C 180,E1 -22972.054,E2 -22972.054} C_VEL
LIN {X 0,Y 180.187,Z 886.888,A -85,B 0,C 180,E1 -22974.483,E2 -22974.483} C_VEL
LIN {X 0,Y 182.295,Z 879.306,A -85,B 0,C 180,E1 -22976.318,E2 -22976.318} C_VEL
LIN {X 0,Y 184.246,Z 871.352,A -85,B 0,C 180,E1 -22977.857,E2 -22977.857} C_VEL
LIN {X 0,Y 185.867,Z 863.129,A -85,B 0,C 180,E1 -22979.132,E2 -22979.132} C_VEL
LIN {X 0,Y 187.35,Z 854.299,A -85,B 0,C 180,E1 -22980.176,E2 -22980.176} C_VEL
LIN {X 0,Y 188.42,Z 845.141,A -85,B 0,C 180,E1 -22980.987,E2 -22980.987} C_VEL
LIN {X 0,Y 189.095,Z 836.468,A -85,B 0,C 180,E1 -22981.511,E2 -22981.511} C_VEL
LIN {X 0,Y 190.519,Z 803.93,A -85,B 0,C 180,E1 -22982.723,E2 -22982.723} C_VEL
LIN {X 0,Y 186.074,Z 792.511,A -85,B 0,C 180,E1 -22984.134,E2 -22984.134} C_VEL
LIN {X 0,Y 181.592,Z 783.64,A -85,B 0,C 180,E1 -22985.527,E2 -22985.527} C_VEL
LIN {X 0,Y 173.495,Z 770.165,A -85,B 0,C 180,E1 -22988.167,E2 -22988.167} C_VEL
LIN {X 0,Y 171.729,Z 767.468,A -85,B 0,C 180,E1 -22988.795,E2 -22988.795} C_VEL
LIN {X 0,Y 171.403,Z 766.261,A -85,B 0,C 180,E1 -22989.206,E2 -22989.206} C_VEL
LIN {X 0,Y 171.339,Z 765.931,A -85,B 0,C 180,E1 -22991.017,E2 -22991.017} C_VEL
LIN {X 0,Y 171.321,Z 765.893,A -85,B 0,C 180,E1 -22995.782,E2 -22995.782} C_VEL
LIN {X 0,Y 171.358,Z 765.919,A -85,B 0,C 180,E1 -23001.193,E2 -23001.193} C_VEL
LIN {X 0,Y 171.399,Z 765.931,A -85,B 0,C 180,E1 -23005.092,E2 -23005.092} C_VEL
LIN {X 0,Y 171.449,Z 765.942,A -85,B 0,C 180,E1 -23010.534,E2 -23010.534} C_VEL
LIN {X 0,Y 171.446,Z 765.917,A -85,B 0,C 180,E1 -23015.8,E2 -23015.8} C_VEL
LIN {X 0,Y 171.578,Z 765.9,A -85,B 0,C 180,E1 -23020.871,E2 -23020.871} C_VEL
LIN {X 0,Y 171.571,Z 765.914,A -85,B 0,C 180,E1 -23025.772,E2 -23025.772} C_VEL
LIN {X 0,Y 171.902,Z 765.853,A -85,B 0,C 180,E1 -23030.588,E2 -23030.588} C_VEL
LIN {X 0,Y 171.829,Z 765.877,A -85,B 0,C 180,E1 -23035.308,E2 -23035.308} C_VEL
LIN {X 0,Y 172.334,Z 765.805,A -85,B 0,C 180,E1 -23040,E2 -23040} C_VEL
LIN {X 0,Y 171.821,Z 765.868,A -85,B 0,C 180,E1 -23044.692,E2 -23044.692} C_VEL
LIN {X 0,Y 171.888,Z 765.872,A -85,B 0,C 180,E1 -23049.413,E2 -23049.413} C_VEL
LIN {X 0,Y 171.595,Z 765.896,A -85,B 0,C 180,E1 -23054.225,E2 -23054.225} C_VEL
LIN {X 0,Y 171.545,Z 765.904,A -85,B 0,C 180,E1 -23059.562,E2 -23059.562} C_VEL
LIN {X 0,Y 171.47,Z 765.939,A -85,B 0,C 180,E1 -23065.616,E2 -23065.616} C_VEL
LIN {X 0,Y 171.44,Z 765.918,A -85,B 0,C 180,E1 -23070.585,E2 -23070.585} C_VEL
LIN {X 0,Y 171.398,Z 765.922,A -85,B 0,C 180,E1 -23075.033,E2 -23075.033} C_VEL
LIN {X 0,Y 171.376,Z 765.867,A -85,B 0,C 180,E1 -23078.815,E2 -23078.815} C_VEL
LIN {X 0,Y 171.344,Z 765.948,A -85,B 0,C 180,E1 -23084.21,E2 -23084.21} C_VEL
LIN {X 0,Y 171.419,Z 766.143,A -85,B 0,C 180,E1 -23088.461,E2 -23088.461} C_VEL
LIN {X 0,Y 172.352,Z 769.578,A -85,B 0,C 180,E1 -23091.016,E2 -23091.016} C_VEL
LIN {X 0,Y 174.501,Z 773.872,A -85,B 0,C 180,E1 -23091.915,E2 -23091.915} C_VEL
LIN {X 0,Y 180.644,Z 786.234,A -85,B 0,C 180,E1 -23094.012,E2 -23094.012} C_VEL
LIN {X 0,Y 186.842,Z 801.119,A -85,B 0,C 180,E1 -23096.048,E2 -23096.048} C_VEL
LIN {X 0,Y 187.961,Z 805.893,A -85,B 0,C 180,E1 -23096.49,E2 -23096.49} C_VEL
LIN {X 0,Y 189.76,Z 822.514,A -85,B 0,C 180,E1 -23097.578,E2 -23097.578} C_VEL
LIN {X 0,Y 188.571,Z 847.793,A -85,B 0,C 180,E1 -23098.548,E2 -23098.548} C_VEL
LIN {X 0,Y 187.415,Z 858.878,A -85,B 0,C 180,E1 -23099.274,E2 -23099.274} C_VEL
LIN {X 0,Y 185.505,Z 870.512,A -85,B 0,C 180,E1 -23100.494,E2 -23100.494} C_VEL
LIN {X 0,Y 183.666,Z 879.723,A -85,B 0,C 180,E1 -23101.846,E2 -23101.846} C_VEL
LIN {X 0,Y 181.785,Z 887.484,A -85,B 0,C 180,E1 -23103.293,E2 -23103.293} C_VEL
LIN {X 0,Y 179.552,Z 895.336,A -85,B 0,C 180,E1 -23105.116,E2 -23105.116} C_VEL
LIN {X 0,Y 177.351,Z 902.685,A -85,B 0,C 180,E1 -23107.271,E2 -23107.271} C_VEL
LIN {X 0,Y 175.072,Z 909.501,A -85,B 0,C 180,E1 -23109.773,E2 -23109.773} C_VEL
LIN {X 0,Y 173.245,Z 913.023,A -85,B 0,C 180,E1 -23111.218,E2 -23111.218} C_VEL
LIN {X 0,Y 168.749,Z 918.016,A -85,B 0,C 180,E1 -23113.669,E2 -23113.669} C_VEL
LIN {X 0,Y 164.519,Z 922.06,A -85,B 0,C 180,E1 -23116.427,E2 -23116.427} C_VEL
LIN {X 0,Y 163.152,Z 924.091,A -85,B 0,C 180,E1 -23118.312,E2 -23118.312} C_VEL
LIN {X 0,Y 162.637,Z 925.725,A -85,B 0,C 180,E1 -23120.046,E2 -23120.046} C_VEL
LIN {X 0,Y 162.143,Z 927.475,A -85,B 0,C 180,E1 -23122.528,E2 -23122.528} C_VEL
LIN {X 0,Y 161.928,Z 928.73,A -85,B 0,C 180,E1 -23125.02,E2 -23125.02} C_VEL
LIN {X 0,Y 161.836,Z 929.51,A -85,B 0,C 180,E1 -23127.511,E2 -23127.511} C_VEL
LIN {X 0,Y 161.907,Z 929.806,A -85,B 0,C 180,E1 -23130,E2 -23130} C_VEL
LIN {X 0,Y 161.828,Z 929.467,A -85,B 0,C 180,E1 -23132.741,E2 -23132.741} C_VEL
LIN {X 0,Y 162.143,Z 927.428,A -85,B 0,C 180,E1 -23137.472,E2 -23137.472} C_VEL
LIN {X 0,Y 162.993,Z 924.5,A -85,B 0,C 180,E1 -23141.188,E2 -23141.188} C_VEL
LIN {X 0,Y 163.85,Z 921.832,A -85,B 0,C 180,E1 -23143.645,E2 -23143.645} C_VEL
LIN {X 0,Y 165.67,Z 916.626,A -85,B 0,C 180,E1 -23147.275,E2 -23147.275} C_VEL
LIN {X 0,Y 168.206,Z 909.769,A -85,B 0,C 180,E1 -23150.802,E2 -23150.802} C_VEL
LIN {X 0,Y 170.807,Z 902.283,A -85,B 0,C 180,E1 -23153.652,E2 -23153.652} C_VEL
LIN {X 0,Y 173.146,Z 894.9,A -85,B 0,C 180,E1 -23155.871,E2 -23155.871} C_VEL
LIN {X 0,Y 175.498,Z 886.997,A -85,B 0,C 180,E1 -23157.745,E2 -23157.745} C_VEL
LIN {X 0,Y 177.735,Z 877.895,A -85,B 0,C 180,E1 -23159.457,E2 -23159.457} C_VEL
LIN {X 0,Y 179.933,Z 866.804,A -85,B 0,C 180,E1 -23161.004,E2 -23161.004} C_VEL
LIN {X 0,Y 181.576,Z 856.251,A -85,B 0,C 180,E1 -23161.991,E2 -23161.991} C_VEL
LIN {X 0,Y 182.519,Z 846.385,A -85,B 0,C 180,E1 -23162.621,E2 -23162.621} C_VEL
LIN {X 0,Y 183.59,Z 821.78,A -85,B 0,C 180,E1 -23163.601,E2 -23163.601} C_VEL
LIN {X 0,Y 181.592,Z 804.913,A -85,B 0,C 180,E1 -23164.807,E2 -23164.807} C_VEL
LIN {X 0,Y 175.142,Z 789.251,A -85,B 0,C 180,E1 -23167.057,E2 -23167.057} C_VEL
LIN {X 0,Y 169.365,Z 777.599,A -85,B 0,C 180,E1 -23169.154,E2 -23169.154} C_VEL
LIN {X 0,Y 166.685,Z 772.839,A -85,B 0,C 180,E1 -23170.163,E2 -23170.163} C_VEL
LIN {X 0,Y 164.965,Z 769.334,A -85,B 0,C 180,E1 -23170.987,E2 -23170.987} C_VEL
LIN {X 0,Y 164.304,Z 766.891,A -85,B 0,C 180,E1 -23172.949,E2 -23172.949} C_VEL
LIN {X 0,Y 164.292,Z 766.792,A -85,B 0,C 180,E1 -23176.809,E2 -23176.809} C_VEL
LIN {X 0,Y 164.305,Z 766.746,A -85,B 0,C 180,E1 -23180.348,E2 -23180.348} C_VEL
LIN {X 0,Y 164.337,Z 766.785,A -85,B 0,C 180,E1 -23184.346,E2 -23184.346} C_VEL
LIN {X 0,Y 164.39,Z 766.797,A -85,B 0,C 180,E1 -23189.135,E2 -23189.135} C_VEL
LIN {X 0,Y 164.417,Z 766.817,A -85,B 0,C 180,E1 -23194.694,E2 -23194.694} C_VEL
LIN {X 0,Y 164.486,Z 766.779,A -85,B 0,C 180,E1 -23200.051,E2 -23200.051} C_VEL
LIN {X 0,Y 164.544,Z 766.781,A -85,B 0,C 180,E1 -23205.151,E2 -23205.151} C_VEL
LIN {X 0,Y 164.803,Z 766.746,A -85,B 0,C 180,E1 -23210.179,E2 -23210.179} C_VEL
LIN {X 0,Y 164.851,Z 766.764,A -85,B 0,C 180,E1 -23212.652,E2 -23212.652} C_VEL
LIN {X 0,Y 165.05,Z 766.693,A -85,B 0,C 180,E1 -23217.56,E2 -23217.56} C_VEL
LIN {X 0,Y 165.297,Z 766.68,A -85,B 0,C 180,E1 -23220,E2 -23220} C_VEL
LIN {X 0,Y 164.776,Z 766.751,A -85,B 0,C 180,E1 -23224.894,E2 -23224.894} C_VEL
LIN {X 0,Y 164.849,Z 766.719,A -85,B 0,C 180,E1 -23227.348,E2 -23227.348} C_VEL
LIN {X 0,Y 164.741,Z 766.768,A -85,B 0,C 180,E1 -23231.127,E2 -23231.127} C_VEL
LIN {X 0,Y 164.454,Z 766.774,A -85,B 0,C 180,E1 -23237.407,E2 -23237.407} C_VEL
LIN {X 0,Y 164.45,Z 766.798,A -85,B 0,C 180,E1 -23239.992,E2 -23239.992} C_VEL
LIN {X 0,Y 164.386,Z 766.788,A -85,B 0,C 180,E1 -23246.128,E2 -23246.128} C_VEL
LIN {X 0,Y 164.375,Z 766.812,A -85,B 0,C 180,E1 -23251.227,E2 -23251.227} C_VEL
LIN {X 0,Y 164.296,Z 766.833,A -85,B 0,C 180,E1 -23256.79,E2 -23256.79} C_VEL
LIN {X 0,Y 164.291,Z 766.778,A -85,B 0,C 180,E1 -23259.916,E2 -23259.916} C_VEL
LIN {X 0,Y 164.28,Z 766.76,A -85,B 0,C 180,E1 -23263.342,E2 -23263.342} C_VEL
LIN {X 0,Y 164.346,Z 767.042,A -85,B 0,C 180,E1 -23268.911,E2 -23268.911} C_VEL
LIN {X 0,Y 164.607,Z 768.135,A -85,B 0,C 180,E1 -23269.395,E2 -23269.395} C_VEL
LIN {X 0,Y 166.191,Z 770.787,A -85,B 0,C 180,E1 -23270.039,E2 -23270.039} C_VEL
LIN {X 0,Y 167.239,Z 772.201,A -85,B 0,C 180,E1 -23270.42,E2 -23270.42} C_VEL
LIN {X 0,Y 171.995,Z 779.896,A -85,B 0,C 180,E1 -23272.129,E2 -23272.129} C_VEL
LIN {X 0,Y 178.637,Z 791.517,A -85,B 0,C 180,E1 -23274.348,E2 -23274.348} C_VEL
LIN {X 0,Y 182.823,Z 801.167,A -85,B 0,C 180,E1 -23275.743,E2 -23275.743} C_VEL
LIN {X 0,Y 184.441,Z 806.025,A -85,B 0,C 180,E1 -23276.311,E2 -23276.311} C_VEL
LIN {X 0,Y 182.88,Z 837.929,A -85,B 0,C 180,E1 -23277.535,E2 -23277.535} C_VEL
LIN {X 0,Y 182.114,Z 846.87,A -85,B 0,C 180,E1 -23278.131,E2 -23278.131} C_VEL
LIN {X 0,Y 180.635,Z 857.57,A -85,B 0,C 180,E1 -23279.157,E2 -23279.157} C_VEL
LIN {X 0,Y 178.687,Z 867.793,A -85,B 0,C 180,E1 -23280.551,E2 -23280.551} C_VEL
LIN {X 0,Y 176.745,Z 876.427,A -85,B 0,C 180,E1 -23282.146,E2 -23282.146} C_VEL
LIN {X 0,Y 174.427,Z 884.54,A -85,B 0,C 180,E1 -23284.013,E2 -23284.013} C_VEL
LIN {X 0,Y 172.359,Z 891.228,A -85,B 0,C 180,E1 -23285.936,E2 -23285.936} C_VEL
LIN {X 0,Y 170.234,Z 897.562,A -85,B 0,C 180,E1 -23288.188,E2 -23288.188} C_VEL
LIN {X 0,Y 168.353,Z 902.825,A -85,B 0,C 180,E1 -23290.49,E2 -23290.49} C_VEL
LIN {X 0,Y 166.713,Z 907.217,A -85,B 0,C 180,E1 -23292.837,E2 -23292.837} C_VEL
LIN {X 0,Y 164.766,Z 912.38,A -85,B 0,C 180,E1 -23296.432,E2 -23296.432} C_VEL
LIN {X 0,Y 163.768,Z 915.026,A -85,B 0,C 180,E1 -23298.865,E2 -23298.865} C_VEL
LIN {X 0,Y 162.699,Z 917.922,A -85,B 0,C 180,E1 -23302.554,E2 -23302.554} C_VEL
LIN {X 0,Y 162.255,Z 919.182,A -85,B 0,C 180,E1 -23305.03,E2 -23305.03} C_VEL
LIN {X 0,Y 161.998,Z 919.975,A -85,B 0,C 180,E1 -23307.514,E2 -23307.514} C_VEL
LIN {X 0,Y 161.963,Z 920.276,A -85,B 0,C 180,E1 -23310,E2 -23310} C_VEL
LIN {X 0,Y 161.996,Z 919.996,A -85,B 0,C 180,E1 -23312.486,E2 -23312.486} C_VEL
LIN {X 0,Y 162.255,Z 919.245,A -85,B 0,C 180,E1 -23314.97,E2 -23314.97} C_VEL
LIN {X 0,Y 162.693,Z 918.027,A -85,B 0,C 180,E1 -23317.446,E2 -23317.446} C_VEL
LIN {X 0,Y 163.708,Z 915.176,A -85,B 0,C 180,E1 -23321.139,E2 -23321.139} C_VEL
LIN {X 0,Y 164.694,Z 912.578,A -85,B 0,C 180,E1 -23323.574,E2 -23323.574} C_VEL
LIN {X 0,Y 166.651,Z 907.467,A -85,B 0,C 180,E1 -23327.17,E2 -23327.17} C_VEL
LIN {X 0,Y 168.769,Z 901.964,A -85,B 0,C 180,E1 -23330.094,E2 -23330.094} C_VEL
LIN {X 0,Y 171.263,Z 895.041,A -85,B 0,C 180,E1 -23332.945,E2 -23332.945} C_VEL
LIN {X 0,Y 173.772,Z 887.093,A -85,B 0,C 180,E1 -23335.45,E2 -23335.45} C_VEL
LIN {X 0,Y 175.982,Z 879.51,A -85,B 0,C 180,E1 -23337.34,E2 -23337.34} C_VEL
LIN {X 0,Y 178.002,Z 871.556,A -85,B 0,C 180,E1 -23338.925,E2 -23338.925} C_VEL
LIN {X 0,Y 179.718,Z 863.331,A -85,B 0,C 180,E1 -23340.231,E2 -23340.231} C_VEL
LIN {X 0,Y 181.263,Z 854.499,A -85,B 0,C 180,E1 -23341.301,E2 -23341.301} C_VEL
LIN {X 0,Y 182.346,Z 845.548,A -85,B 0,C 180,E1 -23342.12,E2 -23342.12} C_VEL
LIN {X 0,Y 183.094,Z 836.66,A -85,B 0,C 180,E1 -23342.669,E2 -23342.669} C_VEL
LIN {X 0,Y 184.571,Z 805.763,A -85,B 0,C 180,E1 -23343.841,E2 -23343.841} C_VEL
LIN {X 0,Y 179.579,Z 793.261,A -85,B 0,C 180,E1 -23345.525,E2 -23345.525} C_VEL
LIN {X 0,Y 172.8,Z 781.185,A -85,B 0,C 180,E1 -23347.778,E2 -23347.778} C_VEL
LIN {X 0,Y 168.695,Z 774.622,A -85,B 0,C 180,E1 -23349.228,E2 -23349.228} C_VEL
LIN {X 0,Y 166.441,Z 771.091,A -85,B 0,C 180,E1 -23350.063,E2 -23350.063} C_VEL
LIN {X 0,Y 164.812,Z 768.706,A -85,B 0,C 180,E1 -23350.689,E2 -23350.689} C_VEL
LIN {X 0,Y 164.385,Z 767.25,A -85,B 0,C 180,E1 -23351.104,E2 -23351.104} C_VEL
LIN {X 0,Y 164.294,Z 766.868,A -85,B 0,C 180,E1 -23351.533,E2 -23351.533} C_VEL
LIN {X 0,Y 164.263,Z 766.763,A -85,B 0,C 180,E1 -23356.799,E2 -23356.799} C_VEL
LIN {X 0,Y 164.296,Z 766.78,A -85,B 0,C 180,E1 -23360.352,E2 -23360.352} C_VEL
LIN {X 0,Y 164.331,Z 766.82,A -85,B 0,C 180,E1 -23364.349,E2 -23364.349} C_VEL
LIN {X 0,Y 164.39,Z 766.813,A -85,B 0,C 180,E1 -23369.134,E2 -23369.134} C_VEL
LIN {X 0,Y 164.407,Z 766.786,A -85,B 0,C 180,E1 -23374.692,E2 -23374.692} C_VEL
LIN {X 0,Y 164.485,Z 766.794,A -85,B 0,C 180,E1 -23380.051,E2 -23380.051} C_VEL
LIN {X 0,Y 164.501,Z 766.784,A -85,B 0,C 180,E1 -23385.147,E2 -23385.147} C_VEL
LIN {X 0,Y 164.814,Z 766.74,A -85,B 0,C 180,E1 -23390.179,E2 -23390.179} C_VEL
LIN {X 0,Y 164.86,Z 766.718,A -85,B 0,C 180,E1 -23392.652,E2 -23392.652} C_VEL
LIN {X 0,Y 165.054,Z 766.737,A -85,B 0,C 180,E1 -23397.559,E2 -23397.559} C_VEL
LIN {X 0,Y 165.297,Z 766.68,A -85,B 0,C 180,E1 -23400,E2 -23400} C_VEL
LIN {X 0,Y 164.77,Z 766.748,A -85,B 0,C 180,E1 -23404.893,E2 -23404.893} C_VEL
LIN {X 0,Y 164.851,Z 766.764,A -85,B 0,C 180,E1 -23407.348,E2 -23407.348} C_VEL
LIN {X 0,Y 164.743,Z 766.739,A -85,B 0,C 180,E1 -23411.131,E2 -23411.131} C_VEL
LIN {X 0,Y 164.507,Z 766.805,A -85,B 0,C 180,E1 -23417.4,E2 -23417.4} C_VEL
LIN {X 0,Y 164.474,Z 766.779,A -85,B 0,C 180,E1 -23419.989,E2 -23419.989} C_VEL
LIN {X 0,Y 164.394,Z 766.818,A -85,B 0,C 180,E1 -23426.133,E2 -23426.133} C_VEL
LIN {X 0,Y 164.374,Z 766.804,A -85,B 0,C 180,E1 -23431.227,E2 -23431.227} C_VEL
LIN {X 0,Y 164.305,Z 766.765,A -85,B 0,C 180,E1 -23436.786,E2 -23436.786} C_VEL
LIN {X 0,Y 164.301,Z 766.747,A -85,B 0,C 180,E1 -23439.913,E2 -23439.913} C_VEL
LIN {X 0,Y 164.307,Z 766.796,A -85,B 0,C 180,E1 -23443.352,E2 -23443.352} C_VEL
LIN {X 0,Y 164.326,Z 766.94,A -85,B 0,C 180,E1 -23447.043,E2 -23447.043} C_VEL
LIN {X 0,Y 164.949,Z 769.322,A -85,B 0,C 180,E1 -23448.903,E2 -23448.903} C_VEL
LIN {X 0,Y 167.117,Z 773.471,A -85,B 0,C 180,E1 -23449.894,E2 -23449.894} C_VEL
LIN {X 0,Y 172.389,Z 783.421,A -85,B 0,C 180,E1 -23451.862,E2 -23451.862} C_VEL
LIN {X 0,Y 178.647,Z 797.302,A -85,B 0,C 180,E1 -23454.087,E2 -23454.087} C_VEL
LIN {X 0,Y 181.829,Z 805.802,A -85,B 0,C 180,E1 -23455.206,E2 -23455.206} C_VEL
LIN {X 0,Y 183.752,Z 822.812,A -85,B 0,C 180,E1 -23456.403,E2 -23456.403} C_VEL
LIN {X 0,Y 182.557,Z 847.6,A -85,B 0,C 180,E1 -23457.387,E2 -23457.387} C_VEL
LIN {X 0,Y 181.368,Z 858.679,A -85,B 0,C 180,E1 -23458.132,E2 -23458.132} C_VEL
LIN {X 0,Y 179.371,Z 870.31,A -85,B 0,C 180,E1 -23459.379,E2 -23459.379} C_VEL
LIN {X 0,Y 177.706,Z 878.508,A -85,B 0,C 180,E1 -23460.595,E2 -23460.595} C_VEL
LIN {X 0,Y 175.463,Z 887.278,A -85,B 0,C 180,E1 -23462.249,E2 -23462.249} C_VEL
LIN {X 0,Y 173.136,Z 895.13,A -85,B 0,C 180,E1 -23464.128,E2 -23464.128} C_VEL
LIN {X 0,Y 170.821,Z 902.478,A -85,B 0,C 180,E1 -23466.35,E2 -23466.35} C_VEL
LIN {X 0,Y 168.209,Z 909.932,A -85,B 0,C 180,E1 -23469.198,E2 -23469.198} C_VEL
LIN {X 0,Y 165.671,Z 916.739,A -85,B 0,C 180,E1 -23472.726,E2 -23472.726} C_VEL
LIN {X 0,Y 163.851,Z 921.919,A -85,B 0,C 180,E1 -23476.355,E2 -23476.355} C_VEL
LIN {X 0,Y 163.152,Z 924.091,A -85,B 0,C 180,E1 -23478.312,E2 -23478.312} C_VEL
LIN {X 0,Y 161.929,Z 925.935,A -85,B 0,C 180,E1 -23480.26,E2 -23480.26} C_VEL
LIN {X 0,Y 158.476,Z 928.068,A -85,B 0,C 180,E1 -23483.502,E2 -23483.502} C_VEL
LIN {X 0,Y 155.382,Z 929.257,A -85,B 0,C 180,E1 -23486.932,E2 -23486.932} C_VEL
LIN {X 0,Y 154.751,Z 929.497,A -85,B 0,C 180,E1 -23489.112,E2 -23489.112} C_VEL
LIN {X 0,Y 154.738,Z 929.291,A -85,B 0,C 180,E1 -23492.603,E2 -23492.603} C_VEL
LIN {X 0,Y 154.793,Z 928.491,A -85,B 0,C 180,E1 -23495.21,E2 -23495.21} C_VEL
LIN {X 0,Y 155.083,Z 927.218,A -85,B 0,C 180,E1 -23497.814,E2 -23497.814} C_VEL
LIN {X 0,Y 156.01,Z 924.289,A -85,B 0,C 180,E1 -23501.696,E2 -23501.696} C_VEL
LIN {X 0,Y 156.951,Z 921.622,A -85,B 0,C 180,E1 -23504.258,E2 -23504.258} C_VEL
LIN {X 0,Y 158.877,Z 916.415,A -85,B 0,C 180,E1 -23508.038,E2 -23508.038} C_VEL
LIN {X 0,Y 161.585,Z 909.558,A -85,B 0,C 180,E1 -23511.697,E2 -23511.697} C_VEL
LIN {X 0,Y 164.322,Z 902.072,A -85,B 0,C 180,E1 -23514.646,E2 -23514.646} C_VEL
LIN {X 0,Y 166.787,Z 894.688,A -85,B 0,C 180,E1 -23516.935,E2 -23516.935} C_VEL
LIN {X 0,Y 169.24,Z 886.784,A -85,B 0,C 180,E1 -23518.865,E2 -23518.865} C_VEL
LIN {X 0,Y 171.628,Z 877.471,A -85,B 0,C 180,E1 -23520.663,E2 -23520.663} C_VEL
LIN {X 0,Y 173.88,Z 866.674,A -85,B 0,C 180,E1 -23522.198,E2 -23522.198} C_VEL
LIN {X 0,Y 175.532,Z 856.464,A -85,B 0,C 180,E1 -23523.187,E2 -23523.187} C_VEL
LIN {X 0,Y 176.512,Z 847.141,A -85,B 0,C 180,E1 -23523.813,E2 -23523.813} C_VEL
LIN {X 0,Y 177.697,Z 822.732,A -85,B 0,C 180,E1 -23524.816,E2 -23524.816} C_VEL
LIN {X 0,Y 175.88,Z 807.253,A -85,B 0,C 180,E1 -23525.984,E2 -23525.984} C_VEL
LIN {X 0,Y 169.93,Z 792.655,A -85,B 0,C 180,E1 -23528.205,E2 -23528.205} C_VEL
LIN {X 0,Y 164.434,Z 781.46,A -85,B 0,C 180,E1 -23530.339,E2 -23530.339} C_VEL
LIN {X 0,Y 159.721,Z 773.08,A -85,B 0,C 180,E1 -23532.274,E2 -23532.274} C_VEL
LIN {X 0,Y 157.542,Z 769.021,A -85,B 0,C 180,E1 -23533.39,E2 -23533.39} C_VEL
LIN {X 0,Y 157.223,Z 767.834,A -85,B 0,C 180,E1 -23534.34,E2 -23534.34} C_VEL
LIN {X 0,Y 157.212,Z 767.632,A -85,B 0,C 180,E1 -23539.462,E2 -23539.462} C_VEL
LIN {X 0,Y 157.284,Z 767.664,A -85,B 0,C 180,E1 -23544.488,E2 -23544.488} C_VEL
LIN {X 0,Y 157.293,Z 767.692,A -85,B 0,C 180,E1 -23548.096,E2 -23548.096} C_VEL
LIN {X 0,Y 157.322,Z 767.696,A -85,B 0,C 180,E1 -23553.466,E2 -23553.466} C_VEL
LIN {X 0,Y 157.395,Z 767.659,A -85,B 0,C 180,E1 -23559.668,E2 -23559.668} C_VEL
LIN {X 0,Y 157.473,Z 767.67,A -85,B 0,C 180,E1 -23564.468,E2 -23564.468} C_VEL
LIN {X 0,Y 157.727,Z 767.62,A -85,B 0,C 180,E1 -23569.733,E2 -23569.733} C_VEL
LIN {X 0,Y 157.808,Z 767.641,A -85,B 0,C 180,E1 -23572.322,E2 -23572.322} C_VEL
LIN {X 0,Y 158.259,Z 767.555,A -85,B 0,C 180,E1 -23580,E2 -23580} C_VEL
LIN {X 0,Y 157.726,Z 767.624,A -85,B 0,C 180,E1 -23585.113,E2 -23585.113} C_VEL
LIN {X 0,Y 157.805,Z 767.596,A -85,B 0,C 180,E1 -23587.678,E2 -23587.678} C_VEL
LIN {X 0,Y 157.671,Z 767.65,A -85,B 0,C 180,E1 -23591.297,E2 -23591.297} C_VEL
LIN {X 0,Y 157.425,Z 767.657,A -85,B 0,C 180,E1 -23595.537,E2 -23595.537} C_VEL
LIN {X 0,Y 157.358,Z 767.693,A -85,B 0,C 180,E1 -23600.935,E2 -23600.935} C_VEL
LIN {X 0,Y 157.31,Z 767.671,A -85,B 0,C 180,E1 -23606.681,E2 -23606.681} C_VEL
LIN {X 0,Y 157.276,Z 767.683,A -85,B 0,C 180,E1 -23612.428,E2 -23612.428} C_VEL
LIN {X 0,Y 157.269,Z 767.707,A -85,B 0,C 180,E1 -23616.45,E2 -23616.45} C_VEL
LIN {X 0,Y 157.193,Z 767.641,A -85,B 0,C 180,E1 -23622.117,E2 -23622.117} C_VEL
LIN {X 0,Y 157.285,Z 767.931,A -85,B 0,C 180,E1 -23626.708,E2 -23626.708} C_VEL
LIN {X 0,Y 157.598,Z 769.169,A -85,B 0,C 180,E1 -23627.224,E2 -23627.224} C_VEL
LIN {X 0,Y 159.119,Z 771.723,A -85,B 0,C 180,E1 -23627.908,E2 -23627.908} C_VEL
LIN {X 0,Y 160.175,Z 772.887,A -85,B 0,C 180,E1 -23628.32,E2 -23628.32} C_VEL
LIN {X 0,Y 162.458,Z 776.392,A -85,B 0,C 180,E1 -23629.24,E2 -23629.24} C_VEL
LIN {X 0,Y 169.215,Z 787.432,A -85,B 0,C 180,E1 -23631.788,E2 -23631.788} C_VEL
LIN {X 0,Y 175.016,Z 798.409,A -85,B 0,C 180,E1 -23633.83,E2 -23633.83} C_VEL
LIN {X 0,Y 178.526,Z 807.427,A -85,B 0,C 180,E1 -23635.092,E2 -23635.092} C_VEL
LIN {X 0,Y 176.929,Z 838.23,A -85,B 0,C 180,E1 -23636.305,E2 -23636.305} C_VEL
LIN {X 0,Y 176.214,Z 846.627,A -85,B 0,C 180,E1 -23636.883,E2 -23636.883} C_VEL
LIN {X 0,Y 174.963,Z 855.595,A -85,B 0,C 180,E1 -23637.734,E2 -23637.734} C_VEL
LIN {X 0,Y 173.212,Z 864.464,A -85,B 0,C 180,E1 -23638.847,E2 -23638.847} C_VEL
LIN {X 0,Y 171.243,Z 873.995,A -85,B 0,C 180,E1 -23640.495,E2 -23640.495} C_VEL
LIN {X 0,Y 168.401,Z 883.733,A -85,B 0,C 180,E1 -23642.673,E2 -23642.673} C_VEL
LIN {X 0,Y 165.922,Z 891.439,A -85,B 0,C 180,E1 -23644.94,E2 -23644.94} C_VEL
LIN {X 0,Y 163.666,Z 897.773,A -85,B 0,C 180,E1 -23647.265,E2 -23647.265} C_VEL
LIN {X 0,Y 161.691,Z 903.035,A -85,B 0,C 180,E1 -23649.652,E2 -23649.652} C_VEL
LIN {X 0,Y 159.942,Z 907.427,A -85,B 0,C 180,E1 -23652.086,E2 -23652.086} C_VEL
LIN {X 0,Y 157.871,Z 912.59,A -85,B 0,C 180,E1 -23655.827,E2 -23655.827} C_VEL
LIN {X 0,Y 156.804,Z 915.236,A -85,B 0,C 180,E1 -23658.364,E2 -23658.364} C_VEL
LIN {X 0,Y 155.659,Z 918.132,A -85,B 0,C 180,E1 -23662.215,E2 -23662.215} C_VEL
LIN {X 0,Y 155.092,Z 919.654,A -85,B 0,C 180,E1 -23665.516,E2 -23665.516} C_VEL
LIN {X 0,Y 154.878,Z 920.484,A -85,B 0,C 180,E1 -23670,E2 -23670} C_VEL
LIN {X 0,Y 155.092,Z 919.716,A -85,B 0,C 180,E1 -23674.484,E2 -23674.484} C_VEL
LIN {X 0,Y 155.654,Z 918.235,A -85,B 0,C 180,E1 -23677.785,E2 -23677.785} C_VEL
LIN {X 0,Y 156.754,Z 915.384,A -85,B 0,C 180,E1 -23681.64,E2 -23681.64} C_VEL
LIN {X 0,Y 157.811,Z 912.785,A -85,B 0,C 180,E1 -23684.178,E2 -23684.178} C_VEL
LIN {X 0,Y 159.891,Z 907.674,A -85,B 0,C 180,E1 -23687.92,E2 -23687.92} C_VEL
LIN {X 0,Y 162.139,Z 902.17,A -85,B 0,C 180,E1 -23690.953,E2 -23690.953} C_VEL
LIN {X 0,Y 164.755,Z 895.247,A -85,B 0,C 180,E1 -23693.906,E2 -23693.906} C_VEL
LIN {X 0,Y 167.41,Z 887.297,A -85,B 0,C 180,E1 -23696.49,E2 -23696.49} C_VEL
LIN {X 0,Y 169.728,Z 879.714,A -85,B 0,C 180,E1 -23698.437,E2 -23698.437} C_VEL
LIN {X 0,Y 171.828,Z 871.76,A -85,B 0,C 180,E1 -23700.069,E2 -23700.069} C_VEL
LIN {X 0,Y 173.642,Z 863.533,A -85,B 0,C 180,E1 -23701.406,E2 -23701.406} C_VEL
LIN {X 0,Y 175.25,Z 854.745,A -85,B 0,C 180,E1 -23702.498,E2 -23702.498} C_VEL
LIN {X 0,Y 176.391,Z 845.787,A -85,B 0,C 180,E1 -23703.338,E2 -23703.338} C_VEL
LIN {X 0,Y 177.162,Z 836.938,A -85,B 0,C 180,E1 -23703.902,E2 -23703.902} C_VEL
LIN {X 0,Y 178.615,Z 807.466,A -85,B 0,C 180,E1 -23705.059,E2 -23705.059} C_VEL
LIN {X 0,Y 174.009,Z 796.191,A -85,B 0,C 180,E1 -23706.706,E2 -23706.706} C_VEL
LIN {X 0,Y 166.88,Z 783.415,A -85,B 0,C 180,E1 -23709.26,E2 -23709.26} C_VEL
LIN {X 0,Y 161.971,Z 775.858,A -85,B 0,C 180,E1 -23711.139,E2 -23711.139} C_VEL
LIN {X 0,Y 159.653,Z 772.237,A -85,B 0,C 180,E1 -23712.09,E2 -23712.09} C_VEL
LIN {X 0,Y 157.882,Z 769.866,A -85,B 0,C 180,E1 -23712.823,E2 -23712.823} C_VEL
LIN {X 0,Y 157.3,Z 768.11,A -85,B 0,C 180,E1 -23713.361,E2 -23713.361} C_VEL
LIN {X 0,Y 157.181,Z 767.707,A -85,B 0,C 180,E1 -23714.323,E2 -23714.323} C_VEL
LIN {X 0,Y 157.199,Z 767.65,A -85,B 0,C 180,E1 -23719.467,E2 -23719.467} C_VEL
LIN {X 0,Y 157.279,Z 767.695,A -85,B 0,C 180,E1 -23724.486,E2 -23724.486} C_VEL
LIN {X 0,Y 157.294,Z 767.684,A -85,B 0,C 180,E1 -23728.096,E2 -23728.096} C_VEL
LIN {X 0,Y 157.315,Z 767.67,A -85,B 0,C 180,E1 -23733.465,E2 -23733.465} C_VEL
LIN {X 0,Y 157.393,Z 767.682,A -85,B 0,C 180,E1 -23739.669,E2 -23739.669} C_VEL
LIN {X 0,Y 157.437,Z 767.655,A -85,B 0,C 180,E1 -23744.464,E2 -23744.464} C_VEL
LIN {X 0,Y 157.736,Z 767.627,A -85,B 0,C 180,E1 -23749.734,E2 -23749.734} C_VEL
LIN {X 0,Y 157.817,Z 767.594,A -85,B 0,C 180,E1 -23752.322,E2 -23752.322} C_VEL
LIN {X 0,Y 158.004,Z 767.616,A -85,B 0,C 180,E1 -23757.45,E2 -23757.45} C_VEL
LIN {X 0,Y 158.259,Z 767.555,A -85,B 0,C 180,E1 -23760,E2 -23760} C_VEL
LIN {X 0,Y 157.808,Z 767.64,A -85,B 0,C 180,E1 -23767.678,E2 -23767.678} C_VEL
LIN {X 0,Y 157.674,Z 767.618,A -85,B 0,C 180,E1 -23771.303,E2 -23771.303} C_VEL
LIN {X 0,Y 157.473,Z 767.671,A -85,B 0,C 180,E1 -23775.532,E2 -23775.532} C_VEL
LIN {X 0,Y 157.371,Z 767.659,A -85,B 0,C 180,E1 -23780.932,E2 -23780.932} C_VEL
LIN {X 0,Y 157.315,Z 767.694,A -85,B 0,C 180,E1 -23786.684,E2 -23786.684} C_VEL
LIN {X 0,Y 157.276,Z 767.704,A -85,B 0,C 180,E1 -23792.427,E2 -23792.427} C_VEL
LIN {X 0,Y 157.276,Z 767.644,A -85,B 0,C 180,E1 -23796.453,E2 -23796.453} C_VEL
LIN {X 0,Y 157.213,Z 767.651,A -85,B 0,C 180,E1 -23802.109,E2 -23802.109} C_VEL
LIN {X 0,Y 157.24,Z 767.914,A -85,B 0,C 180,E1 -23805.654,E2 -23805.654} C_VEL
LIN {X 0,Y 157.633,Z 769.234,A -85,B 0,C 180,E1 -23806.587,E2 -23806.587} C_VEL
LIN {X 0,Y 159.999,Z 773.427,A -85,B 0,C 180,E1 -23807.724,E2 -23807.724} C_VEL
LIN {X 0,Y 165.478,Z 783.289,A -85,B 0,C 180,E1 -23809.964,E2 -23809.964} C_VEL
LIN {X 0,Y 171.237,Z 795.595,A -85,B 0,C 180,E1 -23812.195,E2 -23812.195} C_VEL
LIN {X 0,Y 176.138,Z 807.897,A -85,B 0,C 180,E1 -23814.022,E2 -23814.022} C_VEL
LIN {X 0,Y 177.817,Z 823.267,A -85,B 0,C 180,E1 -23815.153,E2 -23815.153} C_VEL
LIN {X 0,Y 176.615,Z 847.407,A -85,B 0,C 180,E1 -23816.145,E2 -23816.145} C_VEL
LIN {X 0,Y 175.397,Z 858.481,A -85,B 0,C 180,E1 -23816.911,E2 -23816.911} C_VEL
LIN {X 0,Y 173.296,Z 870.106,A -85,B 0,C 180,E1 -23818.183,E2 -23818.183} C_VEL
LIN {X 0,Y 171.534,Z 878.303,A -85,B 0,C 180,E1 -23819.426,E2 -23819.426} C_VEL
LIN {X 0,Y 169.216,Z 887.073,A -85,B 0,C 180,E1 -23821.13,E2 -23821.13} C_VEL
LIN {X 0,Y 166.778,Z 894.924,A -85,B 0,C 180,E1 -23823.063,E2 -23823.063} C_VEL
LIN {X 0,Y 164.337,Z 902.272,A -85,B 0,C 180,E1 -23825.357,E2 -23825.357} C_VEL
LIN {X 0,Y 161.593,Z 909.726,A -85,B 0,C 180,E1 -23828.304,E2 -23828.304} C_VEL
LIN {X 0,Y 158.878,Z 916.531,A -85,B 0,C 180,E1 -23831.962,E2 -23831.962} C_VEL
LIN {X 0,Y 156.952,Z 921.711,A -85,B 0,C 180,E1 -23835.743,E2 -23835.743} C_VEL
LIN {X 0,Y 155.642,Z 925.517,A -85,B 0,C 180,E1 -23839.594,E2 -23839.594} C_VEL
LIN {X 0,Y 155.083,Z 927.266,A -85,B 0,C 180,E1 -23842.186,E2 -23842.186} C_VEL
LIN {X 0,Y 154.85,Z 928.522,A -85,B 0,C 180,E1 -23844.792,E2 -23844.792} C_VEL
LIN {X 0,Y 154.751,Z 929.497,A -85,B 0,C 180,E1 -23849.112,E2 -23849.112} C_VEL
LIN {X 0,Y 154.476,Z 929.547,A -85,B 0,C 180,E1 -23850.561,E2 -23850.561} C_VEL
LIN {X 0,Y 153.685,Z 929.394,A -85,B 0,C 180,E1 -23851.992,E2 -23851.992} C_VEL
LIN {X 0,Y 151.334,Z 928.574,A -85,B 0,C 180,E1 -23854.826,E2 -23854.826} C_VEL
LIN {X 0,Y 149.128,Z 927.281,A -85,B 0,C 180,E1 -23857.729,E2 -23857.729} C_VEL
LIN {X 0,Y 148.481,Z 925.94,A -85,B 0,C 180,E1 -23859.963,E2 -23859.963} C_VEL
LIN {X 0,Y 148.589,Z 925.364,A -85,B 0,C 180,E1 -23860.709,E2 -23860.709} C_VEL
LIN {X 0,Y 149.522,Z 922.9,A -85,B 0,C 180,E1 -23863.593,E2 -23863.593} C_VEL
LIN {X 0,Y 151.375,Z 918.128,A -85,B 0,C 180,E1 -23867.565,E2 -23867.565} C_VEL
LIN {X 0,Y 153.445,Z 912.967,A -85,B 0,C 180,E1 -23870.791,E2 -23870.791} C_VEL
LIN {X 0,Y 155.514,Z 907.927,A -85,B 0,C 180,E1 -23873.293,E2 -23873.293} C_VEL
LIN {X 0,Y 157.874,Z 901.859,A -85,B 0,C 180,E1 -23875.724,E2 -23875.724} C_VEL
LIN {X 0,Y 160.492,Z 894.477,A -85,B 0,C 180,E1 -23878.083,E2 -23878.083} C_VEL
LIN {X 0,Y 163.053,Z 886.571,A -85,B 0,C 180,E1 -23880.071,E2 -23880.071} C_VEL
LIN {X 0,Y 165.36,Z 877.984,A -85,B 0,C 180,E1 -23881.786,E2 -23881.786} C_VEL
LIN {X 0,Y 167.889,Z 866.606,A -85,B 0,C 180,E1 -23883.472,E2 -23883.472} C_VEL
LIN {X 0,Y 169.653,Z 856.219,A -85,B 0,C 180,E1 -23884.498,E2 -23884.498} C_VEL
LIN {X 0,Y 170.625,Z 847.279,A -85,B 0,C 180,E1 -23885.122,E2 -23885.122} C_VEL
LIN {X 0,Y 171.811,Z 822.808,A -85,B 0,C 180,E1 -23886.177,E2 -23886.177} C_VEL
LIN {X 0,Y 170.23,Z 809.564,A -85,B 0,C 180,E1 -23887.246,E2 -23887.246} C_VEL
LIN {X 0,Y 164.7,Z 795.932,A -85,B 0,C 180,E1 -23889.459,E2 -23889.459} C_VEL
LIN {X 0,Y 159.669,Z 785.474,A -85,B 0,C 180,E1 -23891.559,E2 -23891.559} C_VEL
LIN {X 0,Y 155.391,Z 777.751,A -85,B 0,C 180,E1 -23893.44,E2 -23893.44} C_VEL
LIN {X 0,Y 152.7,Z 773.23,A -85,B 0,C 180,E1 -23894.687,E2 -23894.687} C_VEL
LIN {X 0,Y 150.729,Z 770.592,A -85,B 0,C 180,E1 -23895.622,E2 -23895.622} C_VEL
LIN {X 0,Y 150.265,Z 769.217,A -85,B 0,C 180,E1 -23896.081,E2 -23896.081} C_VEL
LIN {X 0,Y 150.161,Z 768.66,A -85,B 0,C 180,E1 -23896.67,E2 -23896.67} C_VEL
LIN {X 0,Y 150.177,Z 768.514,A -85,B 0,C 180,E1 -23902.528,E2 -23902.528} C_VEL
LIN {X 0,Y 150.217,Z 768.584,A -85,B 0,C 180,E1 -23907.367,E2 -23907.367} C_VEL
LIN {X 0,Y 150.244,Z 768.567,A -85,B 0,C 180,E1 -23912.719,E2 -23912.719} C_VEL
LIN {X 0,Y 150.352,Z 768.533,A -85,B 0,C 180,E1 -23919.208,E2 -23919.208} C_VEL
LIN {X 0,Y 150.38,Z 768.562,A -85,B 0,C 180,E1 -23923.716,E2 -23923.716} C_VEL
LIN {X 0,Y 150.65,Z 768.496,A -85,B 0,C 180,E1 -23929.246,E2 -23929.246} C_VEL
LIN {X 0,Y 150.743,Z 768.519,A -85,B 0,C 180,E1 -23931.96,E2 -23931.96} C_VEL
LIN {X 0,Y 151.22,Z 768.431,A -85,B 0,C 180,E1 -23940,E2 -23940} C_VEL
LIN {X 0,Y 150.682,Z 768.483,A -85,B 0,C 180,E1 -23947.165,E2 -23947.165} C_VEL
LIN {X 0,Y 150.604,Z 768.532,A -85,B 0,C 180,E1 -23951.486,E2 -23951.486} C_VEL
LIN {X 0,Y 150.332,Z 768.534,A -85,B 0,C 180,E1 -23956.29,E2 -23956.29} C_VEL
LIN {X 0,Y 150.34,Z 768.565,A -85,B 0,C 180,E1 -23960.78,E2 -23960.78} C_VEL
LIN {X 0,Y 150.242,Z 768.554,A -85,B 0,C 180,E1 -23967.28,E2 -23967.28} C_VEL
LIN {X 0,Y 150.215,Z 768.561,A -85,B 0,C 180,E1 -23972.632,E2 -23972.632} C_VEL
LIN {X 0,Y 150.174,Z 768.586,A -85,B 0,C 180,E1 -23977.473,E2 -23977.473} C_VEL
LIN {X 0,Y 150.129,Z 768.519,A -85,B 0,C 180,E1 -23982.92,E2 -23982.92} C_VEL
LIN {X 0,Y 150.202,Z 768.955,A -85,B 0,C 180,E1 -23984.257,E2 -23984.257} C_VEL
LIN {X 0,Y 150.61,Z 770.34,A -85,B 0,C 180,E1 -23984.781,E2 -23984.781} C_VEL
LIN {X 0,Y 152.365,Z 772.896,A -85,B 0,C 180,E1 -23985.627,E2 -23985.627} C_VEL
LIN {X 0,Y 153.341,Z 773.928,A -85,B 0,C 180,E1 -23986.052,E2 -23986.052} C_VEL
LIN {X 0,Y 155.49,Z 777.324,A -85,B 0,C 180,E1 -23987.027,E2 -23987.027} C_VEL
LIN {X 0,Y 160.782,Z 785.402,A -85,B 0,C 180,E1 -23989.243,E2 -23989.243} C_VEL
LIN {X 0,Y 167.691,Z 797.592,A -85,B 0,C 180,E1 -23991.919,E2 -23991.919} C_VEL
LIN {X 0,Y 170.711,Z 804.126,A -85,B 0,C 180,E1 -23993.054,E2 -23993.054} C_VEL
LIN {X 0,Y 172.589,Z 809.051,A -85,B 0,C 180,E1 -23993.775,E2 -23993.775} C_VEL
LIN {X 0,Y 171.063,Z 838.86,A -85,B 0,C 180,E1 -23995.013,E2 -23995.013} C_VEL
LIN {X 0,Y 170.161,Z 848.14,A -85,B 0,C 180,E1 -23995.682,E2 -23995.682} C_VEL
LIN {X 0,Y 168.367,Z 859.511,A -85,B 0,C 180,E1 -23996.871,E2 -23996.871} C_VEL
LIN {X 0,Y 166.478,Z 868.221,A -85,B 0,C 180,E1 -23998.15,E2 -23998.15} C_VEL
LIN {X 0,Y 164.368,Z 876.852,A -85,B 0,C 180,E1 -23999.841,E2 -23999.841} C_VEL
LIN {X 0,Y 161.809,Z 884.963,A -85,B 0,C 180,E1 -24001.813,E2 -24001.813} C_VEL
LIN {X 0,Y 159.54,Z 891.65,A -85,B 0,C 180,E1 -24003.863,E2 -24003.863} C_VEL
LIN {X 0,Y 157.144,Z 897.984,A -85,B 0,C 180,E1 -24006.265,E2 -24006.265} C_VEL
LIN {X 0,Y 155.072,Z 903.246,A -85,B 0,C 180,E1 -24008.742,E2 -24008.742} C_VEL
LIN {X 0,Y 153.212,Z 907.638,A -85,B 0,C 180,E1 -24011.271,E2 -24011.271} C_VEL
LIN {X 0,Y 151.007,Z 912.8,A -85,B 0,C 180,E1 -24015.169,E2 -24015.169} C_VEL
LIN {X 0,Y 149.867,Z 915.445,A -85,B 0,C 180,E1 -24017.817,E2 -24017.817} C_VEL
LIN {X 0,Y 148.634,Z 918.341,A -85,B 0,C 180,E1 -24021.845,E2 -24021.845} C_VEL
LIN {X 0,Y 147.94,Z 920.126,A -85,B 0,C 180,E1 -24026.05,E2 -24026.05} C_VEL
LIN {X 0,Y 147.781,Z 920.693,A -85,B 0,C 180,E1 -24030,E2 -24030} C_VEL
LIN {X 0,Y 147.965,Z 920.139,A -85,B 0,C 180,E1 -24034.084,E2 -24034.084} C_VEL
LIN {X 0,Y 148.629,Z 918.444,A -85,B 0,C 180,E1 -24038.155,E2 -24038.155} C_VEL
LIN {X 0,Y 149.824,Z 915.591,A -85,B 0,C 180,E1 -24042.186,E2 -24042.186} C_VEL
LIN {X 0,Y 150.927,Z 912.993,A -85,B 0,C 180,E1 -24044.839,E2 -24044.839} C_VEL
LIN {X 0,Y 153.153,Z 907.881,A -85,B 0,C 180,E1 -24048.737,E2 -24048.737} C_VEL
LIN {X 0,Y 155.551,Z 902.376,A -85,B 0,C 180,E1 -24051.885,E2 -24051.885} C_VEL
LIN {X 0,Y 158.277,Z 895.454,A -85,B 0,C 180,E1 -24054.95,E2 -24054.95} C_VEL
LIN {X 0,Y 161.104,Z 887.503,A -85,B 0,C 180,E1 -24057.614,E2 -24057.614} C_VEL
LIN {X 0,Y 163.536,Z 879.918,A -85,B 0,C 180,E1 -24059.618,E2 -24059.618} C_VEL
LIN {X 0,Y 165.734,Z 871.963,A -85,B 0,C 180,E1 -24061.296,E2 -24061.296} C_VEL
LIN {X 0,Y 167.644,Z 863.735,A -85,B 0,C 180,E1 -24062.666,E2 -24062.666} C_VEL
LIN {X 0,Y 169.359,Z 854.659,A -85,B 0,C 180,E1 -24063.819,E2 -24063.819} C_VEL
LIN {X 0,Y 170.523,Z 845.954,A -85,B 0,C 180,E1 -24064.648,E2 -24064.648} C_VEL
LIN {X 0,Y 171.332,Z 837.043,A -85,B 0,C 180,E1 -24065.229,E2 -24065.229} C_VEL
LIN {X 0,Y 172.703,Z 809.074,A -85,B 0,C 180,E1 -24066.376,E2 -24066.376} C_VEL
LIN {X 0,Y 168.847,Z 799.783,A -85,B 0,C 180,E1 -24067.842,E2 -24067.842} C_VEL
LIN {X 0,Y 162.202,Z 787.72,A -85,B 0,C 180,E1 -24070.387,E2 -24070.387} C_VEL
LIN {X 0,Y 155.668,Z 777.51,A -85,B 0,C 180,E1 -24073.11,E2 -24073.11} C_VEL
LIN {X 0,Y 153.471,Z 774.218,A -85,B 0,C 180,E1 -24074.098,E2 -24074.098} C_VEL
LIN {X 0,Y 152.51,Z 773.037,A -85,B 0,C 180,E1 -24074.528,E2 -24074.528} C_VEL
LIN {X 0,Y 150.764,Z 770.672,A -85,B 0,C 180,E1 -24075.348,E2 -24075.348} C_VEL
LIN {X 0,Y 150.245,Z 769.089,A -85,B 0,C 180,E1 -24075.865,E2 -24075.865} C_VEL
LIN {X 0,Y 150.125,Z 768.605,A -85,B 0,C 180,E1 -24076.662,E2 -24076.662} C_VEL
LIN {X 0,Y 150.174,Z 768.582,A -85,B 0,C 180,E1 -24082.527,E2 -24082.527} C_VEL
LIN {X 0,Y 150.215,Z 768.561,A -85,B 0,C 180,E1 -24087.368,E2 -24087.368} C_VEL
LIN {X 0,Y 150.242,Z 768.556,A -85,B 0,C 180,E1 -24092.72,E2 -24092.72} C_VEL
LIN {X 0,Y 150.351,Z 768.566,A -85,B 0,C 180,E1 -24099.209,E2 -24099.209} C_VEL
LIN {X 0,Y 150.348,Z 768.532,A -85,B 0,C 180,E1 -24103.712,E2 -24103.712} C_VEL
LIN {X 0,Y 150.656,Z 768.515,A -85,B 0,C 180,E1 -24109.245,E2 -24109.245} C_VEL
LIN {X 0,Y 150.751,Z 768.475,A -85,B 0,C 180,E1 -24111.96,E2 -24111.96} C_VEL
LIN {X 0,Y 151.22,Z 768.431,A -85,B 0,C 180,E1 -24120,E2 -24120} C_VEL
LIN {X 0,Y 150.743,Z 768.519,A -85,B 0,C 180,E1 -24128.04,E2 -24128.04} C_VEL
LIN {X 0,Y 150.607,Z 768.496,A -85,B 0,C 180,E1 -24131.492,E2 -24131.492} C_VEL
LIN {X 0,Y 150.38,Z 768.563,A -85,B 0,C 180,E1 -24136.284,E2 -24136.284} C_VEL
LIN {X 0,Y 150.352,Z 768.533,A -85,B 0,C 180,E1 -24140.792,E2 -24140.792} C_VEL
LIN {X 0,Y 150.244,Z 768.565,A -85,B 0,C 180,E1 -24147.281,E2 -24147.281} C_VEL
LIN {X 0,Y 150.217,Z 768.585,A -85,B 0,C 180,E1 -24152.633,E2 -24152.633} C_VEL
LIN {X 0,Y 150.177,Z 768.512,A -85,B 0,C 180,E1 -24157.472,E2 -24157.472} C_VEL
LIN {X 0,Y 150.151,Z 768.616,A -85,B 0,C 180,E1 -24162.919,E2 -24162.919} C_VEL
LIN {X 0,Y 150.241,Z 769.105,A -85,B 0,C 180,E1 -24163.718,E2 -24163.718} C_VEL
LIN {X 0,Y 151.108,Z 771.342,A -85,B 0,C 180,E1 -24164.463,E2 -24164.463} C_VEL
LIN {X 0,Y 153.669,Z 774.721,A -85,B 0,C 180,E1 -24165.637,E2 -24165.637} C_VEL
LIN {X 0,Y 157.261,Z 781.055,A -85,B 0,C 180,E1 -24167.281,E2 -24167.281} C_VEL
LIN {X 0,Y 161.162,Z 788.268,A -85,B 0,C 180,E1 -24168.959,E2 -24168.959} C_VEL
LIN {X 0,Y 166.714,Z 800.459,A -85,B 0,C 180,E1 -24171.25,E2 -24171.25} C_VEL
LIN {X 0,Y 170.634,Z 810.629,A -85,B 0,C 180,E1 -24172.819,E2 -24172.819} C_VEL
LIN {X 0,Y 171.991,Z 824.652,A -85,B 0,C 180,E1 -24173.87,E2 -24173.87} C_VEL
LIN {X 0,Y 170.769,Z 847.214,A -85,B 0,C 180,E1 -24174.818,E2 -24174.818} C_VEL
LIN {X 0,Y 169.404,Z 858.839,A -85,B 0,C 180,E1 -24175.647,E2 -24175.647} C_VEL
LIN {X 0,Y 167.3,Z 869.903,A -85,B 0,C 180,E1 -24176.9,E2 -24176.9} C_VEL
LIN {X 0,Y 165.494,Z 877.918,A -85,B 0,C 180,E1 -24178.139,E2 -24178.139} C_VEL
LIN {X 0,Y 163.404,Z 885.637,A -85,B 0,C 180,E1 -24179.644,E2 -24179.644} C_VEL
LIN {X 0,Y 160.846,Z 893.696,A -85,B 0,C 180,E1 -24181.629,E2 -24181.629} C_VEL
LIN {X 0,Y 158.486,Z 900.355,A -85,B 0,C 180,E1 -24183.676,E2 -24183.676} C_VEL
LIN {X 0,Y 156.108,Z 906.681,A -85,B 0,C 180,E1 -24186.098,E2 -24186.098} C_VEL
LIN {X 0,Y 153.96,Z 911.937,A -85,B 0,C 180,E1 -24188.581,E2 -24188.581} C_VEL
LIN {X 0,Y 152.122,Z 916.322,A -85,B 0,C 180,E1 -24191.131,E2 -24191.131} C_VEL
LIN {X 0,Y 150.081,Z 921.503,A -85,B 0,C 180,E1 -24195.075,E2 -24195.075} C_VEL
LIN {X 0,Y 148.643,Z 925.309,A -85,B 0,C 180,E1 -24199.098,E2 -24199.098} C_VEL
LIN {X 0,Y 148.038,Z 927.057,A -85,B 0,C 180,E1 -24201.812,E2 -24201.812} C_VEL
LIN {X 0,Y 147.76,Z 928.312,A -85,B 0,C 180,E1 -24204.541,E2 -24204.541} C_VEL
LIN {X 0,Y 147.65,Z 929.219,A -85,B 0,C 180,E1 -24208.329,E2 -24208.329} C_VEL
LIN {X 0,Y 147.716,Z 929.388,A -85,B 0,C 180,E1 -24210,E2 -24210} C_VEL
LIN {X 0,Y 147.644,Z 929.082,A -85,B 0,C 180,E1 -24212.728,E2 -24212.728} C_VEL
LIN {X 0,Y 147.718,Z 928.282,A -85,B 0,C 180,E1 -24215.46,E2 -24215.46} C_VEL
LIN {X 0,Y 148.038,Z 927.008,A -85,B 0,C 180,E1 -24218.188,E2 -24218.188} C_VEL
LIN {X 0,Y 148.589,Z 925.364,A -85,B 0,C 180,E1 -24220.709,E2 -24220.709} C_VEL
LIN {X 0,Y 148.598,Z 923.719,A -85,B 0,C 180,E1 -24222.9,E2 -24222.9} C_VEL
LIN {X 0,Y 147.16,Z 920.211,A -85,B 0,C 180,E1 -24226.459,E2 -24226.459} C_VEL
LIN {X 0,Y 146.182,Z 915.763,A -85,B 0,C 180,E1 -24229.915,E2 -24229.915} C_VEL
LIN {X 0,Y 146.894,Z 912.604,A -85,B 0,C 180,E1 -24231.86,E2 -24231.86} C_VEL
LIN {X 0,Y 149.02,Z 907.716,A -85,B 0,C 180,E1 -24234.372,E2 -24234.372} C_VEL
LIN {X 0,Y 151.478,Z 901.647,A -85,B 0,C 180,E1 -24236.895,E2 -24236.895} C_VEL
LIN {X 0,Y 154.273,Z 894.265,A -85,B 0,C 180,E1 -24239.322,E2 -24239.322} C_VEL
LIN {X 0,Y 156.943,Z 886.358,A -85,B 0,C 180,E1 -24241.371,E2 -24241.371} C_VEL
LIN {X 0,Y 159.706,Z 876.499,A -85,B 0,C 180,E1 -24243.371,E2 -24243.371} C_VEL
LIN {X 0,Y 162.178,Z 865.456,A -85,B 0,C 180,E1 -24244.963,E2 -24244.963} C_VEL
LIN {X 0,Y 163.939,Z 855.397,A -85,B 0,C 180,E1 -24245.951,E2 -24245.951} C_VEL
LIN {X 0,Y 165.009,Z 845.711,A -85,B 0,C 180,E1 -24246.604,E2 -24246.604} C_VEL
LIN {X 0,Y 166.089,Z 823.93,A -85,B 0,C 180,E1 -24247.562,E2 -24247.562} C_VEL
LIN {X 0,Y 164.806,Z 812.316,A -85,B 0,C 180,E1 -24248.532,E2 -24248.532} C_VEL
LIN {X 0,Y 159.356,Z 798.588,A -85,B 0,C 180,E1 -24250.891,E2 -24250.891} C_VEL
LIN {X 0,Y 153.785,Z 787.097,A -85,B 0,C 180,E1 -24253.415,E2 -24253.415} C_VEL
LIN {X 0,Y 148.917,Z 778.645,A -85,B 0,C 180,E1 -24255.767,E2 -24255.767} C_VEL
LIN {X 0,Y 146.534,Z 775.101,A -85,B 0,C 180,E1 -24256.972,E2 -24256.972} C_VEL
LIN {X 0,Y 145.721,Z 774.134,A -85,B 0,C 180,E1 -24257.381,E2 -24257.381} C_VEL
LIN {X 0,Y 143.845,Z 771.787,A -85,B 0,C 180,E1 -24258.365,E2 -24258.365} C_VEL
LIN {X 0,Y 143.217,Z 769.93,A -85,B 0,C 180,E1 -24259.055,E2 -24259.055} C_VEL
LIN {X 0,Y 143.114,Z 769.485,A -85,B 0,C 180,E1 -24259.677,E2 -24259.677} C_VEL
LIN {X 0,Y 143.167,Z 769.465,A -85,B 0,C 180,E1 -24266.566,E2 -24266.566} C_VEL
LIN {X 0,Y 143.19,Z 769.438,A -85,B 0,C 180,E1 -24272.064,E2 -24272.064} C_VEL
LIN {X 0,Y 143.278,Z 769.413,A -85,B 0,C 180,E1 -24278.746,E2 -24278.746} C_VEL
LIN {X 0,Y 143.315,Z 769.446,A -85,B 0,C 180,E1 -24282.889,E2 -24282.889} C_VEL
LIN {X 0,Y 143.595,Z 769.37,A -85,B 0,C 180,E1 -24288.71,E2 -24288.71} C_VEL
LIN {X 0,Y 143.662,Z 769.396,A -85,B 0,C 180,E1 -24291.561,E2 -24291.561} C_VEL
LIN {X 0,Y 144.178,Z 769.306,A -85,B 0,C 180,E1 -24300,E2 -24300} C_VEL
LIN {X 0,Y 143.659,Z 769.359,A -85,B 0,C 180,E1 -24308.44,E2 -24308.44} C_VEL
LIN {X 0,Y 143.549,Z 769.413,A -85,B 0,C 180,E1 -24311.713,E2 -24311.713} C_VEL
LIN {X 0,Y 143.27,Z 769.411,A -85,B 0,C 180,E1 -24317.117,E2 -24317.117} C_VEL
LIN {X 0,Y 143.268,Z 769.45,A -85,B 0,C 180,E1 -24321.245,E2 -24321.245} C_VEL
LIN {X 0,Y 143.19,Z 769.438,A -85,B 0,C 180,E1 -24327.936,E2 -24327.936} C_VEL
LIN {X 0,Y 143.144,Z 769.44,A -85,B 0,C 180,E1 -24333.42,E2 -24333.42} C_VEL
LIN {X 0,Y 143.055,Z 769.421,A -85,B 0,C 180,E1 -24339.692,E2 -24339.692} C_VEL
LIN {X 0,Y 143.157,Z 769.822,A -85,B 0,C 180,E1 -24341.288,E2 -24341.288} C_VEL
LIN {X 0,Y 143.544,Z 771.15,A -85,B 0,C 180,E1 -24341.895,E2 -24341.895} C_VEL
LIN {X 0,Y 145.185,Z 773.597,A -85,B 0,C 180,E1 -24342.811,E2 -24342.811} C_VEL
LIN {X 0,Y 146.384,Z 774.827,A -85,B 0,C 180,E1 -24343.405,E2 -24343.405} C_VEL
LIN {X 0,Y 148.657,Z 778.332,A -85,B 0,C 180,E1 -24344.569,E2 -24344.569} C_VEL
LIN {X 0,Y 154.664,Z 787.22,A -85,B 0,C 180,E1 -24347.356,E2 -24347.356} C_VEL
LIN {X 0,Y 161.434,Z 798.964,A -85,B 0,C 180,E1 -24350.22,E2 -24350.22} C_VEL
LIN {X 0,Y 165.325,Z 806.993,A -85,B 0,C 180,E1 -24351.781,E2 -24351.781} C_VEL
LIN {X 0,Y 166.933,Z 811.536,A -85,B 0,C 180,E1 -24352.46,E2 -24352.46} C_VEL
LIN {X 0,Y 165.34,Z 838.544,A -85,B 0,C 180,E1 -24353.573,E2 -24353.573} C_VEL
LIN {X 0,Y 164.449,Z 847.572,A -85,B 0,C 180,E1 -24354.223,E2 -24354.223} C_VEL
LIN {X 0,Y 162.715,Z 858.474,A -85,B 0,C 180,E1 -24355.349,E2 -24355.349} C_VEL
LIN {X 0,Y 160.5,Z 868.435,A -85,B 0,C 180,E1 -24356.814,E2 -24356.814} C_VEL
LIN {X 0,Y 158.292,Z 877.064,A -85,B 0,C 180,E1 -24358.555,E2 -24358.555} C_VEL
LIN {X 0,Y 155.597,Z 885.175,A -85,B 0,C 180,E1 -24360.58,E2 -24360.58} C_VEL
LIN {X 0,Y 153.22,Z 891.861,A -85,B 0,C 180,E1 -24362.697,E2 -24362.697} C_VEL
LIN {X 0,Y 150.674,Z 898.195,A -85,B 0,C 180,E1 -24365.178,E2 -24365.178} C_VEL
LIN {X 0,Y 148.48,Z 903.456,A -85,B 0,C 180,E1 -24367.749,E2 -24367.749} C_VEL
LIN {X 0,Y 146.508,Z 907.848,A -85,B 0,C 180,E1 -24370.379,E2 -24370.379} C_VEL
LIN {X 0,Y 144.144,Z 913.011,A -85,B 0,C 180,E1 -24374.445,E2 -24374.445} C_VEL
LIN {X 0,Y 142.936,Z 915.655,A -85,B 0,C 180,E1 -24377.217,E2 -24377.217} C_VEL
LIN {X 0,Y 141.607,Z 918.551,A -85,B 0,C 180,E1 -24381.437,E2 -24381.437} C_VEL
LIN {X 0,Y 140.824,Z 920.513,A -85,B 0,C 180,E1 -24386.496,E2 -24386.496} C_VEL
LIN {X 0,Y 140.689,Z 920.902,A -85,B 0,C 180,E1 -24390,E2 -24390} C_VEL
LIN {X 0,Y 140.736,Z 920.622,A -85,B 0,C 180,E1 -24392.862,E2 -24392.862} C_VEL
LIN {X 0,Y 141.076,Z 919.87,A -85,B 0,C 180,E1 -24395.718,E2 -24395.718} C_VEL
LIN {X 0,Y 141.602,Z 918.652,A -85,B 0,C 180,E1 -24398.563,E2 -24398.563} C_VEL
LIN {X 0,Y 142.898,Z 915.799,A -85,B 0,C 180,E1 -24402.787,E2 -24402.787} C_VEL
LIN {X 0,Y 144.076,Z 913.201,A -85,B 0,C 180,E1 -24405.563,E2 -24405.563} C_VEL
LIN {X 0,Y 146.443,Z 908.089,A -85,B 0,C 180,E1 -24409.63,E2 -24409.63} C_VEL
LIN {X 0,Y 148.986,Z 902.583,A -85,B 0,C 180,E1 -24412.903,E2 -24412.903} C_VEL
LIN {X 0,Y 151.874,Z 895.66,A -85,B 0,C 180,E1 -24416.079,E2 -24416.079} C_VEL
LIN {X 0,Y 154.865,Z 887.707,A -85,B 0,C 180,E1 -24418.828,E2 -24418.828} C_VEL
LIN {X 0,Y 157.423,Z 880.123,A -85,B 0,C 180,E1 -24420.891,E2 -24420.891} C_VEL
LIN {X 0,Y 159.729,Z 872.167,A -85,B 0,C 180,E1 -24422.615,E2 -24422.615} C_VEL
LIN {X 0,Y 161.732,Z 863.938,A -85,B 0,C 180,E1 -24424.02,E2 -24424.02} C_VEL
LIN {X 0,Y 163.436,Z 855.397,A -85,B 0,C 180,E1 -24425.138,E2 -24425.138} C_VEL
LIN {X 0,Y 164.664,Z 846.701,A -85,B 0,C 180,E1 -24426.007,E2 -24426.007} C_VEL
LIN {X 0,Y 165.566,Z 837.537,A -85,B 0,C 180,E1 -24426.629,E2 -24426.629} C_VEL
LIN {X 0,Y 167.044,Z 811.289,A -85,B 0,C 180,E1 -24427.711,E2 -24427.711} C_VEL
LIN {X 0,Y 163.795,Z 803.424,A -85,B 0,C 180,E1 -24429.035,E2 -24429.035} C_VEL
LIN {X 0,Y 157.033,Z 791.072,A -85,B 0,C 180,E1 -24431.819,E2 -24431.819} C_VEL
LIN {X 0,Y 151.135,Z 781.923,A -85,B 0,C 180,E1 -24434.462,E2 -24434.462} C_VEL
LIN {X 0,Y 148.783,Z 778.469,A -85,B 0,C 180,E1 -24435.597,E2 -24435.597} C_VEL
LIN {X 0,Y 146.637,Z 775.295,A -85,B 0,C 180,E1 -24436.688,E2 -24436.688} C_VEL
LIN {X 0,Y 145.798,Z 774.168,A -85,B 0,C 180,E1 -24437.121,E2 -24437.121} C_VEL
LIN {X 0,Y 143.86,Z 771.843,A -85,B 0,C 180,E1 -24438.135,E2 -24438.135} C_VEL
LIN {X 0,Y 143.225,Z 770.106,A -85,B 0,C 180,E1 -24438.736,E2 -24438.736} C_VEL
LIN {X 0,Y 143.08,Z 769.484,A -85,B 0,C 180,E1 -24439.668,E2 -24439.668} C_VEL
LIN {X 0,Y 143.088,Z 769.469,A -85,B 0,C 180,E1 -24443.885,E2 -24443.885} C_VEL
LIN {X 0,Y 143.182,Z 769.436,A -85,B 0,C 180,E1 -24447.321,E2 -24447.321} C_VEL
LIN {X 0,Y 143.19,Z 769.44,A -85,B 0,C 180,E1 -24452.064,E2 -24452.064} C_VEL
LIN {X 0,Y 143.276,Z 769.45,A -85,B 0,C 180,E1 -24458.747,E2 -24458.747} C_VEL
LIN {X 0,Y 143.287,Z 769.409,A -85,B 0,C 180,E1 -24462.885,E2 -24462.885} C_VEL
LIN {X 0,Y 143.596,Z 769.403,A -85,B 0,C 180,E1 -24468.71,E2 -24468.71} C_VEL
LIN {X 0,Y 143.67,Z 769.358,A -85,B 0,C 180,E1 -24471.561,E2 -24471.561} C_VEL
LIN {X 0,Y 144.178,Z 769.307,A -85,B 0,C 180,E1 -24480,E2 -24480} C_VEL
LIN {X 0,Y 143.662,Z 769.396,A -85,B 0,C 180,E1 -24488.439,E2 -24488.439} C_VEL
LIN {X 0,Y 143.549,Z 769.374,A -85,B 0,C 180,E1 -24491.712,E2 -24491.712} C_VEL
LIN {X 0,Y 143.315,Z 769.446,A -85,B 0,C 180,E1 -24497.111,E2 -24497.111} C_VEL
LIN {X 0,Y 143.278,Z 769.413,A -85,B 0,C 180,E1 -24501.254,E2 -24501.254} C_VEL
LIN {X 0,Y 143.19,Z 769.437,A -85,B 0,C 180,E1 -24507.936,E2 -24507.936} C_VEL
LIN {X 0,Y 143.167,Z 769.464,A -85,B 0,C 180,E1 -24513.434,E2 -24513.434} C_VEL
LIN {X 0,Y 143.065,Z 769.431,A -85,B 0,C 180,E1 -24519.688,E2 -24519.688} C_VEL
LIN {X 0,Y 143.196,Z 769.942,A -85,B 0,C 180,E1 -24520.788,E2 -24520.788} C_VEL
LIN {X 0,Y 144.01,Z 772.043,A -85,B 0,C 180,E1 -24521.578,E2 -24521.578} C_VEL
LIN {X 0,Y 145.891,Z 774.277,A -85,B 0,C 180,E1 -24522.557,E2 -24522.557} C_VEL
LIN {X 0,Y 149.082,Z 778.764,A -85,B 0,C 180,E1 -24524.172,E2 -24524.172} C_VEL
LIN {X 0,Y 154.598,Z 788.55,A -85,B 0,C 180,E1 -24526.837,E2 -24526.837} C_VEL
LIN {X 0,Y 159.687,Z 799.337,A -85,B 0,C 180,E1 -24529.145,E2 -24529.145} C_VEL
LIN {X 0,Y 164.222,Z 810.559,A -85,B 0,C 180,E1 -24531.11,E2 -24531.11} C_VEL
LIN {X 0,Y 165.254,Z 813.928,A -85,B 0,C 180,E1 -24531.579,E2 -24531.579} C_VEL
LIN {X 0,Y 166.257,Z 825.434,A -85,B 0,C 180,E1 -24532.466,E2 -24532.466} C_VEL
LIN {X 0,Y 165.01,Z 847.021,A -85,B 0,C 180,E1 -24533.396,E2 -24533.396} C_VEL
LIN {X 0,Y 163.703,Z 857.862,A -85,B 0,C 180,E1 -24534.175,E2 -24534.175} C_VEL
LIN {X 0,Y 161.408,Z 869.7,A -85,B 0,C 180,E1 -24535.525,E2 -24535.525} C_VEL
LIN {X 0,Y 159.575,Z 877.471,A -85,B 0,C 180,E1 -24536.748,E2 -24536.748} C_VEL
LIN {X 0,Y 157.319,Z 885.432,A -85,B 0,C 180,E1 -24538.337,E2 -24538.337} C_VEL
LIN {X 0,Y 154.637,Z 893.49,A -85,B 0,C 180,E1 -24540.38,E2 -24540.38} C_VEL
LIN {X 0,Y 152.146,Z 900.149,A -85,B 0,C 180,E1 -24542.489,E2 -24542.489} C_VEL
LIN {X 0,Y 149.637,Z 906.474,A -85,B 0,C 180,E1 -24544.995,E2 -24544.995} C_VEL
LIN {X 0,Y 147.355,Z 911.73,A -85,B 0,C 180,E1 -24547.57,E2 -24547.57} C_VEL
LIN {X 0,Y 145.405,Z 916.115,A -85,B 0,C 180,E1 -24550.224,E2 -24550.224} C_VEL
LIN {X 0,Y 143.215,Z 921.295,A -85,B 0,C 180,E1 -24554.342,E2 -24554.342} C_VEL
LIN {X 0,Y 141.668,Z 925.1,A -85,B 0,C 180,E1 -24558.555,E2 -24558.555} C_VEL
LIN {X 0,Y 141.015,Z 926.849,A -85,B 0,C 180,E1 -24561.401,E2 -24561.401} C_VEL
LIN {X 0,Y 140.696,Z 928.104,A -85,B 0,C 180,E1 -24564.266,E2 -24564.266} C_VEL
LIN {X 0,Y 140.572,Z 929.122,A -85,B 0,C 180,E1 -24569.221,E2 -24569.221} C_VEL
LIN {X 0,Y 140.548,Z 928.873,A -85,B 0,C 180,E1 -24572.866,E2 -24572.866} C_VEL
LIN {X 0,Y 140.645,Z 928.072,A -85,B 0,C 180,E1 -24575.736,E2 -24575.736} C_VEL
LIN {X 0,Y 141.015,Z 926.798,A -85,B 0,C 180,E1 -24578.599,E2 -24578.599} C_VEL
LIN {X 0,Y 142.114,Z 923.869,A -85,B 0,C 180,E1 -24582.858,E2 -24582.858} C_VEL
LIN {X 0,Y 143.214,Z 921.201,A -85,B 0,C 180,E1 -24585.659,E2 -24585.659} C_VEL
LIN {X 0,Y 145.404,Z 915.993,A -85,B 0,C 180,E1 -24589.776,E2 -24589.776} C_VEL
LIN {X 0,Y 146.894,Z 912.604,A -85,B 0,C 180,E1 -24591.86,E2 -24591.86} C_VEL
LIN {X 0,Y 147.74,Z 909.365,A -85,B 0,C 180,E1 -24593.713,E2 -24593.713} C_VEL
LIN {X 0,Y 147.621,Z 903.458,A -85,B 0,C 180,E1 -24596.792,E2 -24596.792} C_VEL
LIN {X 0,Y 147.691,Z 896.859,A -85,B 0,C 180,E1 -24599.691,E2 -24599.691} C_VEL
LIN {X 0,Y 148.755,Z 892.384,A -85,B 0,C 180,E1 -24601.166,E2 -24601.166} C_VEL
LIN {X 0,Y 152.169,Z 882.292,A -85,B 0,C 180,E1 -24603.657,E2 -24603.657} C_VEL
LIN {X 0,Y 154.644,Z 872.768,A -85,B 0,C 180,E1 -24605.41,E2 -24605.41} C_VEL
LIN {X 0,Y 156.797,Z 863.384,A -85,B 0,C 180,E1 -24606.656,E2 -24606.656} C_VEL
LIN {X 0,Y 158.414,Z 853.834,A -85,B 0,C 180,E1 -24607.576,E2 -24607.576} C_VEL
LIN {X 0,Y 159.464,Z 844.188,A -85,B 0,C 180,E1 -24608.199,E2 -24608.199} C_VEL
LIN {X 0,Y 160.436,Z 824.458,A -85,B 0,C 180,E1 -24609.088,E2 -24609.088} C_VEL
LIN {X 0,Y 159.497,Z 815.135,A -85,B 0,C 180,E1 -24609.892,E2 -24609.892} C_VEL
LIN {X 0,Y 154.625,Z 802.59,A -85,B 0,C 180,E1 -24612.169,E2 -24612.169} C_VEL
LIN {X 0,Y 149.486,Z 791.719,A -85,B 0,C 180,E1 -24614.677,E2 -24614.677} C_VEL
LIN {X 0,Y 145.171,Z 783.964,A -85,B 0,C 180,E1 -24616.917,E2 -24616.917} C_VEL
LIN {X 0,Y 142.185,Z 779.684,A -85,B 0,C 180,E1 -24618.526,E2 -24618.526} C_VEL
LIN {X 0,Y 139.922,Z 776.462,A -85,B 0,C 180,E1 -24619.827,E2 -24619.827} C_VEL
LIN {X 0,Y 139.311,Z 775.417,A -85,B 0,C 180,E1 -24620.205,E2 -24620.205} C_VEL
LIN {X 0,Y 137.101,Z 773.239,A -85,B 0,C 180,E1 -24621.495,E2 -24621.495} C_VEL
LIN {X 0,Y 136.153,Z 770.908,A -85,B 0,C 180,E1 -24622.43,E2 -24622.43} C_VEL
LIN {X 0,Y 136.047,Z 770.335,A -85,B 0,C 180,E1 -24623.554,E2 -24623.554} C_VEL
LIN {X 0,Y 136.063,Z 770.325,A -85,B 0,C 180,E1 -24628.901,E2 -24628.901} C_VEL
LIN {X 0,Y 136.147,Z 770.316,A -85,B 0,C 180,E1 -24632.317,E2 -24632.317} C_VEL
LIN {X 0,Y 136.245,Z 770.288,A -85,B 0,C 180,E1 -24638.833,E2 -24638.833} C_VEL
LIN {X 0,Y 136.281,Z 770.296,A -85,B 0,C 180,E1 -24645.058,E2 -24645.058} C_VEL
LIN {X 0,Y 136.498,Z 770.251,A -85,B 0,C 180,E1 -24648.115,E2 -24648.115} C_VEL
LIN {X 0,Y 136.59,Z 770.269,A -85,B 0,C 180,E1 -24651.121,E2 -24651.121} C_VEL
LIN {X 0,Y 137.135,Z 770.182,A -85,B 0,C 180,E1 -24660,E2 -24660} C_VEL
LIN {X 0,Y 136.584,Z 770.242,A -85,B 0,C 180,E1 -24668.88,E2 -24668.88} C_VEL
LIN {X 0,Y 136.492,Z 770.294,A -85,B 0,C 180,E1 -24671.955,E2 -24671.955} C_VEL
LIN {X 0,Y 136.189,Z 770.294,A -85,B 0,C 180,E1 -24678.037,E2 -24678.037} C_VEL
LIN {X 0,Y 136.191,Z 770.333,A -85,B 0,C 180,E1 -24681.74,E2 -24681.74} C_VEL
LIN {X 0,Y 136.1,Z 770.329,A -85,B 0,C 180,E1 -24688.615,E2 -24688.615} C_VEL
LIN {X 0,Y 136.044,Z 770.328,A -85,B 0,C 180,E1 -24694.629,E2 -24694.629} C_VEL
LIN {X 0,Y 136.072,Z 770.64,A -85,B 0,C 180,E1 -24697.773,E2 -24697.773} C_VEL
LIN {X 0,Y 136.441,Z 771.964,A -85,B 0,C 180,E1 -24698.487,E2 -24698.487} C_VEL
LIN {X 0,Y 138.035,Z 774.426,A -85,B 0,C 180,E1 -24699.54,E2 -24699.54} C_VEL
LIN {X 0,Y 139.657,Z 775.921,A -85,B 0,C 180,E1 -24700.462,E2 -24700.462} C_VEL
LIN {X 0,Y 141.707,Z 779.153,A -85,B 0,C 180,E1 -24701.676,E2 -24701.676} C_VEL
LIN {X 0,Y 142.971,Z 780.699,A -85,B 0,C 180,E1 -24702.359,E2 -24702.359} C_VEL
LIN {X 0,Y 148.645,Z 789.165,A -85,B 0,C 180,E1 -24705.293,E2 -24705.293} C_VEL
LIN {X 0,Y 154.15,Z 798.322,A -85,B 0,C 180,E1 -24707.868,E2 -24707.868} C_VEL
LIN {X 0,Y 159.878,Z 809.385,A -85,B 0,C 180,E1 -24710.351,E2 -24710.351} C_VEL
LIN {X 0,Y 161.281,Z 812.979,A -85,B 0,C 180,E1 -24710.969,E2 -24710.969} C_VEL
